// TIA Portal V15 program export: 0 tag tables, 1 data types, 9 data blocks, 101 code blocks (in call order from the OBs), 80 instance data blocks

TYPE "EM_I_OUT_UDT"
// stored: CreationDate 2018-06-03T17:21:19.3788416Z, InterfaceModifiedDate 2018-06-03T17:22:01.3782438Z, IsConsistent true, IsKnowHowProtected false, LibraryConformanceStatus The object is library-conformant., ModifiedDate 2018-06-03T17:22:01.3782438Z
   STRUCT
      Request : Int;
      Command : Int;
      Pressure_SP : REAL;
      placeholder_SP_0 : Byte;   // placeholder
      placeholder_SP_1 : Byte;   // placeholder
      placeholder_SP_2 : Byte;   // placeholder
      placeholder_SP_3 : Byte;   // placeholder
      placeholder_SP_4 : Byte;   // placeholder
      placeholder_SP_5 : Byte;   // placeholder
      placeholder_SP_6 : Byte;   // placeholder
      placeholder_SP_7 : Byte;   // placeholder
      placeholder_SP_8 : Byte;   // placeholder
      placeholder_SP_9 : Byte;   // placeholder
      placeholder_SP_10 : Byte;   // placeholder
      placeholder_SP_11 : Byte;   // placeholder
      placeholder_SP_12 : Byte;   // placeholder
      placeholder_SP_13 : Byte;   // placeholder
      placeholder_SP_14 : Byte;   // placeholder
      placeholder_SP_15 : Byte;   // placeholder
      placeholder_SP_16 : Byte;   // placeholder
      placeholder_SP_17 : Byte;   // placeholder
      placeholder_SP_18 : Byte;   // placeholder
      placeholder_SP_19 : Byte;   // placeholder
      placeholder_SP_20 : Byte;   // placeholder
      placeholder_SP_21 : Byte;   // placeholder
      placeholder_SP_22 : Byte;   // placeholder
      placeholder_SP_23 : Byte;   // placeholder
      placeholder_SP_24 : Byte;   // placeholder
      placeholder_SP_25 : Byte;   // placeholder
      placeholder_SP_26 : Byte;   // placeholder
      placeholder_SP_27 : Byte;   // placeholder
      placeholder_SP_28 : Byte;   // placeholder
      placeholder_SP_29 : Byte;   // placeholder
      placeholder_SP_30 : Byte;   // placeholder
      placeholder_SP_31 : Byte;   // placeholder
      Owner : Int;
      Status : Int;
      CM_error : Bool;
      CM_error_no : DINT;
      q_bACTVIE : Bool;
      Level : REAL;
      Pressure : REAL;
      placeholder_PV_0 : Byte;   // placeholder
      placeholder_PV_1 : Byte;   // placeholder
      placeholder_PV_2 : Byte;   // placeholder
      placeholder_PV_3 : Byte;   // placeholder
      placeholder_PV_4 : Byte;   // placeholder
      placeholder_PV_5 : Byte;   // placeholder
      placeholder_PV_6 : Byte;   // placeholder
      placeholder_PV_7 : Byte;   // placeholder
      placeholder_PV_8 : Byte;   // placeholder
      placeholder_PV_9 : Byte;   // placeholder
      placeholder_PV_10 : Byte;   // placeholder
      placeholder_PV_11 : Byte;   // placeholder
      placeholder_PV_12 : Byte;   // placeholder
      placeholder_PV_13 : Byte;   // placeholder
      placeholder_PV_14 : Byte;   // placeholder
      placeholder_PV_15 : Byte;   // placeholder
      placeholder_PV_16 : Byte;   // placeholder
      placeholder_PV_17 : Byte;   // placeholder
      placeholder_PV_18 : Byte;   // placeholder
      placeholder_PV_19 : Byte;   // placeholder
   END_STRUCT;
END_TYPE

DATA_BLOCK "FIC100_sp"   // DB1
{ S7_Optimized_Access := 'FALSE' }
VERSION : 0.1
// stored: AutoNumber true, CodeModifiedDate 2018-05-31T16:37:51.7325883Z, CompileDate 2018-05-31T16:37:51.7405888Z, CreationDate 2018-05-31T16:36:47.0278874Z, InterfaceModifiedDate 2018-05-31T16:37:42.3500517Z, IsConsistent true, IsKnowHowProtected false, IsOnlyStoredInLoadMemory false, IsPLCDB false, IsWriteProtectedInAS false, ModifiedDate 2018-05-31T16:37:51.7325883Z, ParameterModified 2018-05-31T16:37:42.3500517Z, StructureModified 2018-05-31T16:37:42.3500517Z
   VAR RETAIN
      Operator_Setpoint : Real;
      Set_SP : Bool;
      Output_Value : Real;
      Set_Output : Bool;
   END_VAR
BEGIN
END_DATA_BLOCK

DATA_BLOCK "FIC101_sp"   // DB1
{ S7_Optimized_Access := 'FALSE' }
VERSION : 0.1
// stored: AutoNumber true, CodeModifiedDate 2018-05-31T16:37:51.7325883Z, CompileDate 2018-05-31T16:37:51.7405888Z, CreationDate 2018-05-31T16:36:47.0278874Z, InterfaceModifiedDate 2018-05-31T16:37:42.3500517Z, IsConsistent true, IsKnowHowProtected false, IsOnlyStoredInLoadMemory false, IsPLCDB false, IsWriteProtectedInAS false, ModifiedDate 2018-05-31T16:37:51.7325883Z, ParameterModified 2018-05-31T16:37:42.3500517Z, StructureModified 2018-05-31T16:37:42.3500517Z
   VAR RETAIN
      Operator_Setpoint : Real;
      Set_SP : Bool;
      Output_Value : Real;
      Set_Output : Bool;
   END_VAR
BEGIN
END_DATA_BLOCK

DATA_BLOCK "LIC001_sp"   // DB1
{ S7_Optimized_Access := 'FALSE' }
VERSION : 0.1
// stored: AutoNumber true, CodeModifiedDate 2018-05-31T16:37:51.7325883Z, CompileDate 2018-05-31T16:37:51.7405888Z, CreationDate 2018-05-31T16:36:47.0278874Z, InterfaceModifiedDate 2018-05-31T16:37:42.3500517Z, IsConsistent true, IsKnowHowProtected false, IsOnlyStoredInLoadMemory false, IsPLCDB false, IsWriteProtectedInAS false, ModifiedDate 2018-05-31T16:37:51.7325883Z, ParameterModified 2018-05-31T16:37:42.3500517Z, StructureModified 2018-05-31T16:37:42.3500517Z
   VAR RETAIN
      Operator_Setpoint : Real;
      Set_SP : Bool;
      Output_Value : Real;
      Set_Output : Bool;
   END_VAR
BEGIN
END_DATA_BLOCK

DATA_BLOCK "LIC002_sp"   // DB1
{ S7_Optimized_Access := 'FALSE' }
VERSION : 0.1
// stored: AutoNumber true, CodeModifiedDate 2018-05-31T16:37:51.7325883Z, CompileDate 2018-05-31T16:37:51.7405888Z, CreationDate 2018-05-31T16:36:47.0278874Z, InterfaceModifiedDate 2018-05-31T16:37:42.3500517Z, IsConsistent true, IsKnowHowProtected false, IsOnlyStoredInLoadMemory false, IsPLCDB false, IsWriteProtectedInAS false, ModifiedDate 2018-05-31T16:37:51.7325883Z, ParameterModified 2018-05-31T16:37:42.3500517Z, StructureModified 2018-05-31T16:37:42.3500517Z
   VAR RETAIN
      Operator_Setpoint : Real;
      Set_SP : Bool;
      Output_Value : Real;
      Set_Output : Bool;
   END_VAR
BEGIN
END_DATA_BLOCK

DATA_BLOCK "LIC003_sp"   // DB1
{ S7_Optimized_Access := 'FALSE' }
VERSION : 0.1
// stored: AutoNumber true, CodeModifiedDate 2018-05-31T16:37:51.7325883Z, CompileDate 2018-05-31T16:37:51.7405888Z, CreationDate 2018-05-31T16:36:47.0278874Z, InterfaceModifiedDate 2018-05-31T16:37:42.3500517Z, IsConsistent true, IsKnowHowProtected false, IsOnlyStoredInLoadMemory false, IsPLCDB false, IsWriteProtectedInAS false, ModifiedDate 2018-05-31T16:37:51.7325883Z, ParameterModified 2018-05-31T16:37:42.3500517Z, StructureModified 2018-05-31T16:37:42.3500517Z
   VAR RETAIN
      Operator_Setpoint : Real;
      Set_SP : Bool;
      Output_Value : Real;
      Set_Output : Bool;
   END_VAR
BEGIN
END_DATA_BLOCK

DATA_BLOCK "LIC004_sp"   // DB1
{ S7_Optimized_Access := 'FALSE' }
VERSION : 0.1
// stored: AutoNumber true, CodeModifiedDate 2018-05-31T16:37:51.7325883Z, CompileDate 2018-05-31T16:37:51.7405888Z, CreationDate 2018-05-31T16:36:47.0278874Z, InterfaceModifiedDate 2018-05-31T16:37:42.3500517Z, IsConsistent true, IsKnowHowProtected false, IsOnlyStoredInLoadMemory false, IsPLCDB false, IsWriteProtectedInAS false, ModifiedDate 2018-05-31T16:37:51.7325883Z, ParameterModified 2018-05-31T16:37:42.3500517Z, StructureModified 2018-05-31T16:37:42.3500517Z
   VAR RETAIN
      Operator_Setpoint : Real;
      Set_SP : Bool;
      Output_Value : Real;
      Set_Output : Bool;
   END_VAR
BEGIN
END_DATA_BLOCK

DATA_BLOCK "LIC005_sp"   // DB1
{ S7_Optimized_Access := 'FALSE' }
VERSION : 0.1
// stored: AutoNumber true, CodeModifiedDate 2018-05-31T16:37:51.7325883Z, CompileDate 2018-05-31T16:37:51.7405888Z, CreationDate 2018-05-31T16:36:47.0278874Z, InterfaceModifiedDate 2018-05-31T16:37:42.3500517Z, IsConsistent true, IsKnowHowProtected false, IsOnlyStoredInLoadMemory false, IsPLCDB false, IsWriteProtectedInAS false, ModifiedDate 2018-05-31T16:37:51.7325883Z, ParameterModified 2018-05-31T16:37:42.3500517Z, StructureModified 2018-05-31T16:37:42.3500517Z
   VAR RETAIN
      Operator_Setpoint : Real;
      Set_SP : Bool;
      Output_Value : Real;
      Set_Output : Bool;
   END_VAR
BEGIN
END_DATA_BLOCK

DATA_BLOCK "LIC006_sp"   // DB1
{ S7_Optimized_Access := 'FALSE' }
VERSION : 0.1
// stored: AutoNumber true, CodeModifiedDate 2018-05-31T16:37:51.7325883Z, CompileDate 2018-05-31T16:37:51.7405888Z, CreationDate 2018-05-31T16:36:47.0278874Z, InterfaceModifiedDate 2018-05-31T16:37:42.3500517Z, IsConsistent true, IsKnowHowProtected false, IsOnlyStoredInLoadMemory false, IsPLCDB false, IsWriteProtectedInAS false, ModifiedDate 2018-05-31T16:37:51.7325883Z, ParameterModified 2018-05-31T16:37:42.3500517Z, StructureModified 2018-05-31T16:37:42.3500517Z
   VAR RETAIN
      Operator_Setpoint : Real;
      Set_SP : Bool;
      Output_Value : Real;
      Set_Output : Bool;
   END_VAR
BEGIN
END_DATA_BLOCK

DATA_BLOCK "EM_Index"   // DB2
{ S7_Optimized_Access := 'FALSE' }
VERSION : 0.1
// stored: AutoNumber true, CodeModifiedDate 2018-06-04T11:31:36.2595073Z, CompileDate 2018-06-04T11:31:36.8205394Z, CreationDate 2018-06-04T11:30:27.8755959Z, InterfaceModifiedDate 2018-06-04T11:31:33.0593242Z, IsConsistent true, IsKnowHowProtected false, IsOnlyStoredInLoadMemory false, IsPLCDB false, IsWriteProtectedInAS false, ModifiedDate 2018-06-04T11:31:36.2595073Z, ParameterModified 2018-06-04T11:31:33.0593242Z, StructureModified 2018-06-04T11:31:33.0593242Z
   VAR RETAIN
      DB_Numbers : Array[0..990] of Int;   // DB numbers of the EMs
   END_VAR
BEGIN
END_DATA_BLOCK

ORGANIZATION_BLOCK "Main"   // OB1, STL, ProgramCycle
TITLE = "Main Program Sweep (Cycle)"
{ S7_Optimized_Access := 'FALSE' }
VERSION : 0.1
// stored: AutoNumber false, CodeModifiedDate 2018-06-08T08:01:58.298282Z, CompileDate 2018-06-08T08:01:58.2972819Z, CreationDate 2018-05-29T13:31:39.8908501Z, InterfaceModifiedDate 2007-08-03T16:55:08.419547Z, IsConsistent true, IsKnowHowProtected false, IsWriteProtected false, ModifiedDate 2018-06-08T08:01:58.298282Z, ParameterModified 2007-08-03T16:55:08.419547Z, StructureModified 2007-08-03T16:55:08.419547Z
   VAR_TEMP
      OB1_EV_CLASS : Byte;   // Bits 0-3 = 1 (Coming event), Bits 4-7 = 1 (Event class 1)
      OB1_SCAN_1 : Byte;   // 1 (Cold restart scan 1 of OB 1), 3 (Scan 2-n of OB 1)
      OB1_PRIORITY : Byte;   // Priority of OB Execution
      OB1_OB_NUMBR : Byte;   // 1 (Organization block 1, OB1)
      OB1_RESERVED_1 : Byte;   // Reserved for system
      OB1_RESERVED_2 : Byte;   // Reserved for system
      OB1_PREV_CYCLE : Int;   // Cycle time of previous OB1 scan (milliseconds)
      OB1_MIN_CYCLE : Int;   // Minimum cycle time of OB1 (milliseconds)
      OB1_MAX_CYCLE : Int;   // Maximum cycle time of OB1 (milliseconds)
      OB1_DATE_TIME : Date_And_Time;   // Date and time OB1 started
   END_VAR
BEGIN

NETWORK
TITLE = Main
// comment


      CALL  "Main_Program";


END_ORGANIZATION_BLOCK

FUNCTION "Main_Program" : Void   // FC1, STL
TITLE = Program
{ S7_Optimized_Access := 'TRUE' }
VERSION : 0.1
// Main Program
// stored: AutoNumber true, UDAEnableTagReadback false
BEGIN

NETWORK
TITLE = Main
// comment


      CALL  "Units";

      CALL  "CM_VALVE"
      ( AUT_OP   := ,
        FB_OPEN  := ,
        FB_CLOSE := ,
        QOPEN    := ,
        QCLOSE   := ,
        QMON_ERR := ,
        QCMD_OP  := 
      );



END_FUNCTION

FUNCTION "Units" : Void   // FC1, STL
TITLE = Program
{ S7_Optimized_Access := 'TRUE' }
VERSION : 0.1
// Call all the Units
// stored: AutoNumber true, UDAEnableTagReadback false
BEGIN

NETWORK
TITLE = Main
// comment


// code



END_FUNCTION

FUNCTION_BLOCK "EM_I_OUT"   // FB1, STL
TITLE = EM_I_OUT_fc
{ S7_Optimized_Access := 'TRUE' }
VERSION : 0.1
// EM_I_OUT
// stored: AutoNumber true, UDAEnableTagReadback false
   VAR_INPUT
      sampletime : Real;   // the scantime of this EM/phase, used to increase timers
      em_id : Int;   // undefined - undefined
      Request : Int;   // undefined - undefined
      Command : Int;   // undefined - undefined
      Pressure_SP : REAL;   // undefined - undefined
      Pump_RUN : Bool;   // undefined - undefined
      Pump_QERR : BOOL;   // undefined - General Error
      Pump_EERR : BOOL;   // undefined - External Error
      FS01_PV : Bool;   // Flow Switch - Digital Measurement
      PIC01_PV : REAL;   // Pressure Controller - undefined
      PIC01_ERR : BOOL;   // Pressure Controller - undefined
      LT01_PV : Real;   // Level Transmitter (m) - undefined
      LT01_AHH : Bool;   // Level Transmitter (m) - undefined
      LT01_AH : Bool;   // Level Transmitter (m) - undefined
      LT01_AL : Bool;   // Level Transmitter (m) - undefined
      LT01_ALL : Bool;   // Level Transmitter (m) - undefined
      LT01_ERR : BOOL;   // Level Transmitter (m) - undefined
      XV_Bottom_OPN : BOOL;   // Automatic Bottom Valve - undefined
      XV_Bottom_CLS : BOOL;   // Automatic Bottom Valve - undefined
      XV_Bottom_MERR : BOOL;   // Automatic Bottom Valve - undefined
      BV_Bottom_OPN : BOOL;   // Manual Bottom Valve - undefined
      BV_Bottom_CLS : BOOL;   // Manual Bottom Valve - undefined
      BV_Bottom_MERR : BOOL;   // Manual Bottom Valve - undefined
      BV_Tran_M04_OPN : BOOL;   // Trnasfer Valve to M04 - undefined
      BV_Tran_M04_CLS : BOOL;   // Trnasfer Valve to M04 - undefined
      BV_Tran_M04_MERR : BOOL;   // Trnasfer Valve to M04 - undefined
   END_VAR
   VAR_OUTPUT
      steptime_s : Real;   // complete steptime in seconds. same value as the other steptimes
      steptime_m : Real;   // complete steptime in minutes. same value as the other steptimes
      steptime_h : Real;   // complete steptime in hours. same value as the other steptimes
      first_scan : Bool;   // first scan of the step active
      last_scan : Bool;   // last scan of the step active
      error_index_db : Bool;   // em_id doesn't fit in the index db
      Owner : Int;   // undefined - undefined
      Status : Int;   // undefined - undefined
      CM_error : Bool;   // undefined - undefined
      CM_error_no : DINT;   // undefined - undefined
      q_bACTVIE : Bool;   // undefined - undefined
      Level : REAL;   // undefined - undefined
      Pressure : REAL;   // undefined - undefined
      Pump_ON : Bool;   // undefined - Switch Motor ON
      Pump_AUT : Bool;   // undefined - Swtich Motor to AUTO
      PIC01_EXT : Bool;   // Pressure Controller - Switch to External Mode
      PIC01_SP : Real;   // Pressure Controller - Operator Setpoint in Internal Mode
      PIC01_AUT : Bool;   // Pressure Controller - Switch to Auto Mode
      PIC01_VAL_OUT : Real;   // Pressure Controller - Operator Output Value
      PIC01_SET_SP : Bool;   // Pressure Controller - undefined
      PIC01_SET_OUT : Bool;   // Pressure Controller - undefined
      XV_Bottom_CMD : BOOL;   // Automatic Bottom Valve - Auto command from program
      BV_Bottom_CMD : BOOL;   // Manual Bottom Valve - Auto command from program
      BV_Tran_M04_CMD : BOOL;   // Trnasfer Valve to M04 - Auto command from program
   END_VAR
   VAR DB_SPECIFIC
      previous_Command : Int;   // previous Command
      SP_PV : "EM_I_OUT_UDT";   // UDT for receiving Setpoints and sending Process Values
   END_VAR
   VAR_TEMP
      initial_scan : Bool;   // pulse active on the first cycle of a new scan
      T_dbnum : Int;   // DB number of this block
      T_address : Int;   // address in the Index Table DB
      T_length : Int;   // length of the Index Table DB
   END_VAR
BEGIN

NETWORK
TITLE = Publish DB number to EM Index
// The EM will publish its DB number to the EM Index table


//### 0] init
      CLR;
      =     #error_index_db;


//### 1] Check if the ID of this EM fits inside the EM Index table

      OPN   "EM_Index";  //Open data block as shared data block
      L     DBLG;  //Load length of shared data block (length of DB)
      T     #T_length;  //transfer length to length

      L     #T_length;  //length=length/2
      L     2;
      /I;
      T     #T_length;

// Error and end the block if id bigger than length of the DB
      L     #T_length;
      L     #em_id;
      <=D;
      =     #error_index_db;
      BEC;  //if id is bigger than length end the block

//### 2] Write this DB number to the EM Index table

// find the number of the current fb
      L     DINO;
      T     #T_dbnum;  //find the db number of current fb

// calculate the real address
      L     #em_id;
      L     2;
      *I;
      T     #T_address;

// prepare the pointer for the location in the EM Index DB
// todo: can this code not simpeler? Probably no need to add with the zero-pointer
      OPN   "EM_Index";
      L     P#DBX0.0;
      L     #T_address;
      SLD   3;
      +D;
      LAR1;

//write the DB number to the real address
      L     #T_dbnum;
      T     DBW [AR1, P#0.0];





NETWORK
TITLE = Copy all Setpoints from the UDT
// network comment





      L     #SP_PV.Request;
      T     #Request;



      L     #SP_PV.Command;
      T     #Command;



      L     #SP_PV.Pressure_SP;
      T     #Pressure_SP;




NETWORK
TITLE = Acquiring logic
// network comment


      L     #Request;
      T     #Owner;



NETWORK
TITLE = Steptimers
// If the previous Command is not the same as the current one
// then reset the timers, else increase them
// This is at the start of the FB because normal commandchanges will take
// till the next cycle to become active


// check if Command == previous_Command
      L     #Command;
      L     #previous_Command;
      ==I;  //if condition true then {
      JCN   TIM1;

// increase timer
      L     #sampletime;
      L     #steptime_s;
      +R;
      T     #steptime_s;

      JU    TIM2;
TIM1: NOP   0;

// reset timer
      L     0.0;
      T     #steptime_s;

TIM2: NOP   0;  //end if

// calculate the other two timers
      L     #steptime_s;
      L     60.0;
      /R;
      T     #steptime_m;

      L     60.0;
      /R;
      T     #steptime_h;



NETWORK
TITLE = detect initial scan
// create a pulse active on the first cycle of a new scan
// this signal can be used in the state to execute some actions in the first cycle of the state


      L     #Command;
      L     #previous_Command;
      <>I;
      =     #initial_scan;



NETWORK
TITLE = Save old step
// network comment


      L     #Command;
      T     #previous_Command;



NETWORK
TITLE = Collect the errors from the CMs
// network comment


      CLR;
      O     #Pump_QERR;
      O     #Pump_EERR;
      O     #PIC01_ERR;
      O     #LT01_ERR;
      O     #XV_Bottom_MERR;
      O     #BV_Bottom_MERR;
      O     #BV_Tran_M04_MERR;
      =     #CM_error;



NETWORK
TITLE = Assign a message number to each error
// This code tries to assign an error message to each CM error
// If multiple CMs have an error then it only stores one
// This is the EM type so we don't know which CM instance is connected
// So the error only contains the general name of the CM instance
// If the actual name needs to be shown then it could be deducted
// at a higher level using the CM name and EM instance 
// network_end.render(lib, "ssign a message number to each error") }}


      CLR;

// clear the error no
      L     0;
      T     #CM_error_no;



      A     #Pump_QERR;
      JCN   E1;

      L     50;  //'CM error: Pump_QERR'
      T     #CM_error_no;

E1:   NOP   0;

      A     #Pump_EERR;
      JCN   E2;

      L     51;  //'CM error: Pump_EERR'
      T     #CM_error_no;

E2:   NOP   0;

      A     #PIC01_ERR;
      JCN   E3;

      L     52;  //'CM error: PIC01_ERR'
      T     #CM_error_no;

E3:   NOP   0;

      A     #LT01_ERR;
      JCN   E4;

      L     53;  //'CM error: LT01_ERR'
      T     #CM_error_no;

E4:   NOP   0;

      A     #XV_Bottom_MERR;
      JCN   E5;

      L     54;  //'CM error: XV_Bottom_MERR'
      T     #CM_error_no;

E5:   NOP   0;

      A     #BV_Bottom_MERR;
      JCN   E6;

      L     55;  //'CM error: BV_Bottom_MERR'
      T     #CM_error_no;

E6:   NOP   0;

      A     #BV_Tran_M04_MERR;
      JCN   E7;

      L     56;  //'CM error: BV_Tran_M04_MERR'
      T     #CM_error_no;

E7:   NOP   0;



NETWORK
TITLE = START OF THE STATES
// ################################
// ################################
// 	Placeholder network to indicate the start of the actual sequence
// ################################	  
// ################################


// empty placeholder network



NETWORK
TITLE = State 0: undefined


// skip this network if stepnumber not equal to 0
      L     #Command;
      L     0;
      ==I;
      JCN   J1;

//---------------------------------
// Actions (continuous)
//---------------------------------

// Action: stop Pump
      CLR;
      =     #Pump_ON;

// Action: close XV_Bottom
      CLR;
      =     #XV_Bottom_CMD;

// Action: close BV_Bottom
      CLR;
      =     #BV_Bottom_CMD;

// Action: close BV_Tran_M04
      CLR;
      =     #BV_Tran_M04_CMD;
//---------------------------------
// --- CONDITIONS ---
//---------------------------------

// Condition Logic
      SET;  //make sure RLO is high so the state can happen when no conditions present

      A     #XV_Bottom_CLS;  //XV_Bottom close
      A     #BV_Bottom_CLS;  //BV_Bottom close
      A     #BV_Tran_M04_CLS;  //BV_Tran_M04 close
      JCN   L1;

      L     #Command;
      T     #Status;

L1:   NOP   0;

D1:   NOP   0;

//---------------------------------
// End of network: jump here if step not active
// Jump to end of this FB if the step has been active to avoid
// execution of another step in the same scan
//---------------------------------
      JU    ENDS;
J1:   NOP   0;




NETWORK
TITLE = State 1: undefined


// skip this network if stepnumber not equal to 1
      L     #Command;
      L     1;
      ==I;
      JCN   J2;

//---------------------------------
// Actions (continuous)
//---------------------------------

// Action: stop Pump
      CLR;
      =     #Pump_ON;

// Action: open XV_Bottom
      SET;
      =     #XV_Bottom_CMD;
//---------------------------------
// --- CONDITIONS ---
//---------------------------------

// Condition Logic
      SET;  //make sure RLO is high so the state can happen when no conditions present

      A     #XV_Bottom_OPN;  //XV_Bottom open
      JCN   L2;

      L     #Command;
      T     #Status;

L2:   NOP   0;

D2:   NOP   0;

//---------------------------------
// End of network: jump here if step not active
// Jump to end of this FB if the step has been active to avoid
// execution of another step in the same scan
//---------------------------------
      JU    ENDS;
J2:   NOP   0;




NETWORK
TITLE = State 2: undefined


// skip this network if stepnumber not equal to 2
      L     #Command;
      L     2;
      ==I;
      JCN   J3;

//---------------------------------
// Actions (first scan)
//---------------------------------
      A     #initial_scan;
      JCN   C3;
      L     -1.0;  //value to show that the EM is in a state transition
      T     #Status;

// Action: PIC01_SP = 10.0
      L     10.0;
      T     #PIC01_SP;

// Action: PIC01_SET_SP = true
      SET;
      =     #PIC01_SET_SP;

      JU    D3;
C3:   NOP   0;


//---------------------------------
// Actions (continuous)
//---------------------------------

// Action: start Pump
      SET;
      =     #Pump_ON;

// Action: auto 10.0 bar PIC01
      SET;
      =     #PIC01_AUT;

// Action: open XV_Bottom
      SET;
      =     #XV_Bottom_CMD;

// Action: PIC01_SET_SP = false
      CLR;
      =     #PIC01_SET_SP;
//---------------------------------
// --- CONDITIONS ---
//---------------------------------

// Condition Logic
      SET;  //make sure RLO is high so the state can happen when no conditions present

      A     #Pump_RUN;  //Pump start
      A     #XV_Bottom_OPN;  //XV_Bottom open
      JCN   L3;

      L     #Command;
      T     #Status;

L3:   NOP   0;

D3:   NOP   0;

//---------------------------------
// End of network: jump here if step not active
// Jump to end of this FB if the step has been active to avoid
// execution of another step in the same scan
//---------------------------------
      JU    ENDS;
J3:   NOP   0;




NETWORK
TITLE = State 3: undefined


// skip this network if stepnumber not equal to 3
      L     #Command;
      L     3;
      ==I;
      JCN   J4;

//---------------------------------
// Actions (continuous)
//---------------------------------

// Action: stop Pump
      CLR;
      =     #Pump_ON;

// Action: open BV_Bottom
      SET;
      =     #BV_Bottom_CMD;

// Action: open BV_Tran_M04
      SET;
      =     #BV_Tran_M04_CMD;
//---------------------------------
// --- CONDITIONS ---
//---------------------------------

// Condition Logic
      SET;  //make sure RLO is high so the state can happen when no conditions present

      A     #BV_Bottom_OPN;  //BV_Bottom open
      A     #BV_Tran_M04_OPN;  //BV_Tran_M04 open
      JCN   L4;

      L     #Command;
      T     #Status;

L4:   NOP   0;

D4:   NOP   0;

//---------------------------------
// End of network: jump here if step not active
// Jump to end of this FB if the step has been active to avoid
// execution of another step in the same scan
//---------------------------------
      JU    ENDS;
J4:   NOP   0;




NETWORK
TITLE = State 4: undefined


// skip this network if stepnumber not equal to 4
      L     #Command;
      L     4;
      ==I;
      JCN   J5;

//---------------------------------
// Actions (first scan)
//---------------------------------
      A     #initial_scan;
      JCN   C5;
      L     -1.0;  //value to show that the EM is in a state transition
      T     #Status;

// Action: PIC01_SP = Pressure_SP
      L     #Pressure_SP;
      T     #PIC01_SP;

// Action: PIC01_SET_SP = true
      SET;
      =     #PIC01_SET_SP;

      JU    D5;
C5:   NOP   0;


//---------------------------------
// Actions (continuous)
//---------------------------------

// Action: start Pump
      SET;
      =     #Pump_ON;

// Action: auto Pressure_SP PIC01
      SET;
      =     #PIC01_AUT;

// Action: open BV_Bottom
      SET;
      =     #BV_Bottom_CMD;

// Action: open BV_Tran_M04
      SET;
      =     #BV_Tran_M04_CMD;

// Action: PIC01_SET_SP = false
      CLR;
      =     #PIC01_SET_SP;
//---------------------------------
// --- CONDITIONS ---
//---------------------------------

// Condition Logic
      SET;  //make sure RLO is high so the state can happen when no conditions present

      A     #Pump_RUN;  //Pump start
      A     #BV_Bottom_OPN;  //BV_Bottom open
      A     #BV_Tran_M04_OPN;  //BV_Tran_M04 open
      JCN   L5;

      L     #Command;
      T     #Status;

L5:   NOP   0;

D5:   NOP   0;

//---------------------------------
// End of network: jump here if step not active
// Jump to end of this FB if the step has been active to avoid
// execution of another step in the same scan
//---------------------------------
      JU    ENDS;
J5:   NOP   0;




NETWORK
TITLE = State 5: undefined


// skip this network if stepnumber not equal to 5
      L     #Command;
      L     5;
      ==I;
      JCN   J6;

//---------------------------------
// Actions (first scan)
//---------------------------------
      A     #initial_scan;
      JCN   C6;
      L     -1.0;  //value to show that the EM is in a state transition
      T     #Status;

// Action: PIC01_VAL_OUT = 20.0
      L     20.0;
      T     #PIC01_VAL_OUT;

// Action: PIC01_SET_OUT = true
      SET;
      =     #PIC01_SET_OUT;

      JU    D6;
C6:   NOP   0;


//---------------------------------
// Actions (continuous)
//---------------------------------

// Action: start Pump
      SET;
      =     #Pump_ON;

// Action: manual 20.0 Hz PIC01
      CLR;
      =     #PIC01_AUT;

// Action: open XV_Bottom
      SET;
      =     #XV_Bottom_CMD;

// Action: PIC01_SET_OUT = false
      CLR;
      =     #PIC01_SET_OUT;
//---------------------------------
// --- CONDITIONS ---
//---------------------------------

// Condition Logic
      SET;  //make sure RLO is high so the state can happen when no conditions present

      A     #Pump_RUN;  //Pump start
      A     #XV_Bottom_OPN;  //XV_Bottom open
      JCN   L6;

      L     #Command;
      T     #Status;

L6:   NOP   0;

D6:   NOP   0;

//---------------------------------
// End of network: jump here if step not active
// Jump to end of this FB if the step has been active to avoid
// execution of another step in the same scan
//---------------------------------
      JU    ENDS;
J6:   NOP   0;




NETWORK
TITLE = END OF THE STATES
// ################################
// ################################
// 	Placeholder network to indicate the end of the actual sequence
// ################################	  
// ################################


// jump location for the state that is currently active
ENDS: NOP   0;



NETWORK
TITLE = eneral Actions - After
// General Actions - After


// Action: Level = LT01
      L     #LT01_PV;
      T     #Level;

// Action: Pressure = PIC01
      L     #PIC01_PV;
      T     #Pressure;


NETWORK
TITLE = Copy all Process Values to the UDT
// network comment





      L     #Owner;
      T     #SP_PV.Owner;



      L     #Status;
      T     #SP_PV.Status;



      A     #CM_error;
      =     #SP_PV.CM_error;



      L     #CM_error_no;
      T     #SP_PV.CM_error_no;



      A     #q_bACTVIE;
      =     #SP_PV.q_bACTVIE;



      L     #Level;
      T     #SP_PV.Level;



      L     #Pressure;
      T     #SP_PV.Pressure;




NETWORK
TITLE = Clean up request
// Phases don't clean up their requests on the EM side
// So at the end of the EM reset the request
// If the phase is still there then it will write the request again by the next scan


      L     0;
      T     "request";



NETWORK
TITLE = network title
// network comment


// empty placeholder network


END_FUNCTION_BLOCK

FUNCTION "EM_Instance_10_fc" : Void   // FC1, STL
TITLE = _fc
{ S7_Optimized_Access := 'TRUE' }
VERSION : 0.1
// test
// stored: AutoNumber true, UDAEnableTagReadback false
BEGIN

NETWORK
TITLE = Main
// comment:


// Call the EM FB with the corresponding DB instance
      CALL  "EM_I_OUT", "EM_Instance_10"
      ( sampletime       := ,
        em_id            := 35,
        Request          := ,
        Command          := ,
        Pressure_SP      := ,
        Pump_RUN         := "M106".QNOFF2,
        Pump_QERR        := "M106".QERR,
        Pump_EERR        := "M106".QERR_EXT,
        FS01_PV          := "LS002".QON,
        PIC01_PV         := "FIC101".PV,
        PIC01_ERR        := "FIC101".QERR,
        LT01_PV          := "LT101".QfVal,
        LT01_AHH         := "LT101".LIM_Qb01,
        LT01_AH          := "LT101".LIM_Qb02,
        LT01_AL          := "LT101".LIM_Qb03,
        LT01_ALL         := "LT101".LIM_Qb04,
        LT01_ERR         := "LT101".QERR,
        XV_Bottom_OPN    := ,
        XV_Bottom_CLS    := ,
        XV_Bottom_MERR   := ,
        BV_Bottom_OPN    := "MV007".QOPEN,
        BV_Bottom_CLS    := "MV007".QCLOSE,
        BV_Bottom_MERR   := "MV007".QMON_ERR,
        BV_Tran_M04_OPN  := ,
        BV_Tran_M04_CLS  := ,
        BV_Tran_M04_MERR := ,
        steptime_s       := ,
        steptime_m       := ,
        steptime_h       := ,
        first_scan       := ,
        last_scan        := ,
        error_index_db   := ,
        Owner            := ,
        Status           := ,
        CM_error         := ,
        CM_error_no      := ,
        q_bACTVIE        := ,
        Level            := ,
        Pressure         := ,
        Pump_ON          := "M106".L_ON,
        Pump_AUT         := "M106".L_AUT,
        PIC01_EXT        := "FIC101".L_REMOTE,
        PIC01_SP         := "FIC101".HMI_SP_INT,
        PIC01_AUT        := "FIC101".L_AUT,
        PIC01_VAL_OUT    := "FIC101".HMI_MAN,
        PIC01_SET_SP     := "FIC101".Set_SP,
        PIC01_SET_OUT    := "FIC101".Set_Output,
        XV_Bottom_CMD    := ,
        BV_Bottom_CMD    := "MV007".AUT_OP,
        BV_Tran_M04_CMD  := 
      );
END_FUNCTION

FUNCTION "EM_Instance_11_fc" : Void   // FC1, STL
TITLE = _fc
{ S7_Optimized_Access := 'TRUE' }
VERSION : 0.1
// test
// stored: AutoNumber true, UDAEnableTagReadback false
BEGIN

NETWORK
TITLE = Main
// comment:


// Call the EM FB with the corresponding DB instance
      CALL  "EM_I_OUT", "EM_Instance_11"
      ( sampletime       := ,
        em_id            := 36,
        Request          := ,
        Command          := ,
        Pressure_SP      := ,
        Pump_RUN         := "M106".QNOFF2,
        Pump_QERR        := "M106".QERR,
        Pump_EERR        := "M106".QERR_EXT,
        FS01_PV          := "LS002".QON,
        PIC01_PV         := "FIC101".PV,
        PIC01_ERR        := "FIC101".QERR,
        LT01_PV          := "LT201".QfVal,
        LT01_AHH         := "LT201".LIM_Qb01,
        LT01_AH          := "LT201".LIM_Qb02,
        LT01_AL          := "LT201".LIM_Qb03,
        LT01_ALL         := "LT201".LIM_Qb04,
        LT01_ERR         := "LT201".QERR,
        XV_Bottom_OPN    := "XV001".QOPEN,
        XV_Bottom_CLS    := "XV001".QCLOSE,
        XV_Bottom_MERR   := "XV001".QMON_ERR,
        BV_Bottom_OPN    := ,
        BV_Bottom_CLS    := ,
        BV_Bottom_MERR   := ,
        BV_Tran_M04_OPN  := ,
        BV_Tran_M04_CLS  := ,
        BV_Tran_M04_MERR := ,
        steptime_s       := ,
        steptime_m       := ,
        steptime_h       := ,
        first_scan       := ,
        last_scan        := ,
        error_index_db   := ,
        Owner            := ,
        Status           := ,
        CM_error         := ,
        CM_error_no      := ,
        q_bACTVIE        := ,
        Level            := ,
        Pressure         := ,
        Pump_ON          := "M106".L_ON,
        Pump_AUT         := "M106".L_AUT,
        PIC01_EXT        := "FIC101".L_REMOTE,
        PIC01_SP         := "FIC101".HMI_SP_INT,
        PIC01_AUT        := "FIC101".L_AUT,
        PIC01_VAL_OUT    := "FIC101".HMI_MAN,
        PIC01_SET_SP     := "FIC101".Set_SP,
        PIC01_SET_OUT    := "FIC101".Set_Output,
        XV_Bottom_CMD    := "XV001".AUT_OP,
        BV_Bottom_CMD    := ,
        BV_Tran_M04_CMD  := 
      );
END_FUNCTION

FUNCTION "EM_Instance_12_fc" : Void   // FC1, STL
TITLE = _fc
{ S7_Optimized_Access := 'TRUE' }
VERSION : 0.1
// test
// stored: AutoNumber true, UDAEnableTagReadback false
BEGIN

NETWORK
TITLE = Main
// comment:


// Call the EM FB with the corresponding DB instance
      CALL  "EM_I_OUT", "EM_Instance_12"
      ( sampletime       := ,
        em_id            := 37,
        Request          := ,
        Command          := ,
        Pressure_SP      := ,
        Pump_RUN         := "M106".QNOFF2,
        Pump_QERR        := "M106".QERR,
        Pump_EERR        := "M106".QERR_EXT,
        FS01_PV          := "LS002".QON,
        PIC01_PV         := "FIC101".PV,
        PIC01_ERR        := "FIC101".QERR,
        LT01_PV          := "LT201".QfVal,
        LT01_AHH         := "LT201".LIM_Qb01,
        LT01_AH          := "LT201".LIM_Qb02,
        LT01_AL          := "LT201".LIM_Qb03,
        LT01_ALL         := "LT201".LIM_Qb04,
        LT01_ERR         := "LT201".QERR,
        XV_Bottom_OPN    := "XV002".QOPEN,
        XV_Bottom_CLS    := "XV002".QCLOSE,
        XV_Bottom_MERR   := "XV002".QMON_ERR,
        BV_Bottom_OPN    := ,
        BV_Bottom_CLS    := ,
        BV_Bottom_MERR   := ,
        BV_Tran_M04_OPN  := ,
        BV_Tran_M04_CLS  := ,
        BV_Tran_M04_MERR := ,
        steptime_s       := ,
        steptime_m       := ,
        steptime_h       := ,
        first_scan       := ,
        last_scan        := ,
        error_index_db   := ,
        Owner            := ,
        Status           := ,
        CM_error         := ,
        CM_error_no      := ,
        q_bACTVIE        := ,
        Level            := ,
        Pressure         := ,
        Pump_ON          := "M106".L_ON,
        Pump_AUT         := "M106".L_AUT,
        PIC01_EXT        := "FIC101".L_REMOTE,
        PIC01_SP         := "FIC101".HMI_SP_INT,
        PIC01_AUT        := "FIC101".L_AUT,
        PIC01_VAL_OUT    := "FIC101".HMI_MAN,
        PIC01_SET_SP     := "FIC101".Set_SP,
        PIC01_SET_OUT    := "FIC101".Set_Output,
        XV_Bottom_CMD    := "XV002".AUT_OP,
        BV_Bottom_CMD    := ,
        BV_Tran_M04_CMD  := 
      );
END_FUNCTION

FUNCTION "EM_Instance_13_fc" : Void   // FC1, STL
TITLE = _fc
{ S7_Optimized_Access := 'TRUE' }
VERSION : 0.1
// test
// stored: AutoNumber true, UDAEnableTagReadback false
BEGIN

NETWORK
TITLE = Main
// comment:


// Call the EM FB with the corresponding DB instance
      CALL  "EM_I_OUT", "EM_Instance_13"
      ( sampletime       := ,
        em_id            := 38,
        Request          := ,
        Command          := ,
        Pressure_SP      := ,
        Pump_RUN         := "M106".QNOFF2,
        Pump_QERR        := "M106".QERR,
        Pump_EERR        := "M106".QERR_EXT,
        FS01_PV          := "LS002".QON,
        PIC01_PV         := "FIC101".PV,
        PIC01_ERR        := "FIC101".QERR,
        LT01_PV          := "LT201".QfVal,
        LT01_AHH         := "LT201".LIM_Qb01,
        LT01_AH          := "LT201".LIM_Qb02,
        LT01_AL          := "LT201".LIM_Qb03,
        LT01_ALL         := "LT201".LIM_Qb04,
        LT01_ERR         := "LT201".QERR,
        XV_Bottom_OPN    := "XV003".QOPEN,
        XV_Bottom_CLS    := "XV003".QCLOSE,
        XV_Bottom_MERR   := "XV003".QMON_ERR,
        BV_Bottom_OPN    := ,
        BV_Bottom_CLS    := ,
        BV_Bottom_MERR   := ,
        BV_Tran_M04_OPN  := ,
        BV_Tran_M04_CLS  := ,
        BV_Tran_M04_MERR := ,
        steptime_s       := ,
        steptime_m       := ,
        steptime_h       := ,
        first_scan       := ,
        last_scan        := ,
        error_index_db   := ,
        Owner            := ,
        Status           := ,
        CM_error         := ,
        CM_error_no      := ,
        q_bACTVIE        := ,
        Level            := ,
        Pressure         := ,
        Pump_ON          := "M106".L_ON,
        Pump_AUT         := "M106".L_AUT,
        PIC01_EXT        := "FIC101".L_REMOTE,
        PIC01_SP         := "FIC101".HMI_SP_INT,
        PIC01_AUT        := "FIC101".L_AUT,
        PIC01_VAL_OUT    := "FIC101".HMI_MAN,
        PIC01_SET_SP     := "FIC101".Set_SP,
        PIC01_SET_OUT    := "FIC101".Set_Output,
        XV_Bottom_CMD    := "XV003".AUT_OP,
        BV_Bottom_CMD    := ,
        BV_Tran_M04_CMD  := 
      );
END_FUNCTION

FUNCTION "EM_Instance_14_fc" : Void   // FC1, STL
TITLE = _fc
{ S7_Optimized_Access := 'TRUE' }
VERSION : 0.1
// test
// stored: AutoNumber true, UDAEnableTagReadback false
BEGIN

NETWORK
TITLE = Main
// comment:


// Call the EM FB with the corresponding DB instance
      CALL  "EM_I_OUT", "EM_Instance_14"
      ( sampletime       := ,
        em_id            := 39,
        Request          := ,
        Command          := ,
        Pressure_SP      := ,
        Pump_RUN         := "M106".QNOFF2,
        Pump_QERR        := "M106".QERR,
        Pump_EERR        := "M106".QERR_EXT,
        FS01_PV          := "LS002".QON,
        PIC01_PV         := "FIC101".PV,
        PIC01_ERR        := "FIC101".QERR,
        LT01_PV          := "LT201".QfVal,
        LT01_AHH         := "LT201".LIM_Qb01,
        LT01_AH          := "LT201".LIM_Qb02,
        LT01_AL          := "LT201".LIM_Qb03,
        LT01_ALL         := "LT201".LIM_Qb04,
        LT01_ERR         := "LT201".QERR,
        XV_Bottom_OPN    := "XV004".QOPEN,
        XV_Bottom_CLS    := "XV004".QCLOSE,
        XV_Bottom_MERR   := "XV004".QMON_ERR,
        BV_Bottom_OPN    := ,
        BV_Bottom_CLS    := ,
        BV_Bottom_MERR   := ,
        BV_Tran_M04_OPN  := ,
        BV_Tran_M04_CLS  := ,
        BV_Tran_M04_MERR := ,
        steptime_s       := ,
        steptime_m       := ,
        steptime_h       := ,
        first_scan       := ,
        last_scan        := ,
        error_index_db   := ,
        Owner            := ,
        Status           := ,
        CM_error         := ,
        CM_error_no      := ,
        q_bACTVIE        := ,
        Level            := ,
        Pressure         := ,
        Pump_ON          := "M106".L_ON,
        Pump_AUT         := "M106".L_AUT,
        PIC01_EXT        := "FIC101".L_REMOTE,
        PIC01_SP         := "FIC101".HMI_SP_INT,
        PIC01_AUT        := "FIC101".L_AUT,
        PIC01_VAL_OUT    := "FIC101".HMI_MAN,
        PIC01_SET_SP     := "FIC101".Set_SP,
        PIC01_SET_OUT    := "FIC101".Set_Output,
        XV_Bottom_CMD    := "XV004".AUT_OP,
        BV_Bottom_CMD    := ,
        BV_Tran_M04_CMD  := 
      );
END_FUNCTION

FUNCTION "EM_Instance_1_fc" : Void   // FC1, STL
TITLE = _fc
{ S7_Optimized_Access := 'TRUE' }
VERSION : 0.1
// test
// stored: AutoNumber true, UDAEnableTagReadback false
BEGIN

NETWORK
TITLE = Main
// comment:


// Call the EM FB with the corresponding DB instance
      CALL  "EM_I_OUT", "EM_Instance_1"
      ( sampletime       := ,
        em_id            := 26,
        Request          := ,
        Command          := ,
        Pressure_SP      := ,
        Pump_RUN         := "M100".QNOFF2,
        Pump_QERR        := "M100".QERR,
        Pump_EERR        := "M100".QERR_EXT,
        FS01_PV          := "LS001".QON,
        PIC01_PV         := "LIC001".PV,
        PIC01_ERR        := "LIC001".QERR,
        LT01_PV          := "LT001".QfVal,
        LT01_AHH         := "LT001".LIM_Qb01,
        LT01_AH          := "LT001".LIM_Qb02,
        LT01_AL          := "LT001".LIM_Qb03,
        LT01_ALL         := "LT001".LIM_Qb04,
        LT01_ERR         := "LT001".QERR,
        XV_Bottom_OPN    := ,
        XV_Bottom_CLS    := ,
        XV_Bottom_MERR   := ,
        BV_Bottom_OPN    := "MV001".QOPEN,
        BV_Bottom_CLS    := "MV001".QCLOSE,
        BV_Bottom_MERR   := "MV001".QMON_ERR,
        BV_Tran_M04_OPN  := "MV003".QOPEN,
        BV_Tran_M04_CLS  := "MV003".QCLOSE,
        BV_Tran_M04_MERR := "MV003".QMON_ERR,
        steptime_s       := ,
        steptime_m       := ,
        steptime_h       := ,
        first_scan       := ,
        last_scan        := ,
        error_index_db   := ,
        Owner            := ,
        Status           := ,
        CM_error         := ,
        CM_error_no      := ,
        q_bACTVIE        := ,
        Level            := ,
        Pressure         := ,
        Pump_ON          := "M100".L_ON,
        Pump_AUT         := "M100".L_AUT,
        PIC01_EXT        := "LIC001".L_REMOTE,
        PIC01_SP         := "LIC001".HMI_SP_INT,
        PIC01_AUT        := "LIC001".L_AUT,
        PIC01_VAL_OUT    := "LIC001".HMI_MAN,
        PIC01_SET_SP     := "LIC001".Set_SP,
        PIC01_SET_OUT    := "LIC001".Set_Output,
        XV_Bottom_CMD    := ,
        BV_Bottom_CMD    := "MV001".AUT_OP,
        BV_Tran_M04_CMD  := "MV003".AUT_OP
      );
END_FUNCTION

FUNCTION "EM_Instance_2_fc" : Void   // FC1, STL
TITLE = _fc
{ S7_Optimized_Access := 'TRUE' }
VERSION : 0.1
// test
// stored: AutoNumber true, UDAEnableTagReadback false
BEGIN

NETWORK
TITLE = Main
// comment:


// Call the EM FB with the corresponding DB instance
      CALL  "EM_I_OUT", "EM_Instance_2"
      ( sampletime       := ,
        em_id            := 27,
        Request          := ,
        Command          := ,
        Pressure_SP      := ,
        Pump_RUN         := "M101".QNOFF2,
        Pump_QERR        := "M101".QERR,
        Pump_EERR        := "M101".QERR_EXT,
        FS01_PV          := "LS002".QON,
        PIC01_PV         := "LIC002".PV,
        PIC01_ERR        := "LIC002".QERR,
        LT01_PV          := "LT002".QfVal,
        LT01_AHH         := "LT002".LIM_Qb01,
        LT01_AH          := "LT002".LIM_Qb02,
        LT01_AL          := "LT002".LIM_Qb03,
        LT01_ALL         := "LT002".LIM_Qb04,
        LT01_ERR         := "LT002".QERR,
        XV_Bottom_OPN    := ,
        XV_Bottom_CLS    := ,
        XV_Bottom_MERR   := ,
        BV_Bottom_OPN    := "MV002".QOPEN,
        BV_Bottom_CLS    := "MV002".QCLOSE,
        BV_Bottom_MERR   := "MV002".QMON_ERR,
        BV_Tran_M04_OPN  := "MV003".QOPEN,
        BV_Tran_M04_CLS  := "MV003".QCLOSE,
        BV_Tran_M04_MERR := "MV003".QMON_ERR,
        steptime_s       := ,
        steptime_m       := ,
        steptime_h       := ,
        first_scan       := ,
        last_scan        := ,
        error_index_db   := ,
        Owner            := ,
        Status           := ,
        CM_error         := ,
        CM_error_no      := ,
        q_bACTVIE        := ,
        Level            := ,
        Pressure         := ,
        Pump_ON          := "M101".L_ON,
        Pump_AUT         := "M101".L_AUT,
        PIC01_EXT        := "LIC002".L_REMOTE,
        PIC01_SP         := "LIC002".HMI_SP_INT,
        PIC01_AUT        := "LIC002".L_AUT,
        PIC01_VAL_OUT    := "LIC002".HMI_MAN,
        PIC01_SET_SP     := "LIC002".Set_SP,
        PIC01_SET_OUT    := "LIC002".Set_Output,
        XV_Bottom_CMD    := ,
        BV_Bottom_CMD    := "MV002".AUT_OP,
        BV_Tran_M04_CMD  := "MV003".AUT_OP
      );
END_FUNCTION

FUNCTION "EM_Instance_3_fc" : Void   // FC1, STL
TITLE = _fc
{ S7_Optimized_Access := 'TRUE' }
VERSION : 0.1
// test
// stored: AutoNumber true, UDAEnableTagReadback false
BEGIN

NETWORK
TITLE = Main
// comment:


// Call the EM FB with the corresponding DB instance
      CALL  "EM_I_OUT", "EM_Instance_3"
      ( sampletime       := ,
        em_id            := 28,
        Request          := ,
        Command          := ,
        Pressure_SP      := ,
        Pump_RUN         := "M102".QNOFF2,
        Pump_QERR        := "M102".QERR,
        Pump_EERR        := "M102".QERR_EXT,
        FS01_PV          := "LS002".QON,
        PIC01_PV         := "LIC003".PV,
        PIC01_ERR        := "LIC003".QERR,
        LT01_PV          := "LT003".QfVal,
        LT01_AHH         := "LT003".LIM_Qb01,
        LT01_AH          := "LT003".LIM_Qb02,
        LT01_AL          := "LT003".LIM_Qb03,
        LT01_ALL         := "LT003".LIM_Qb04,
        LT01_ERR         := "LT003".QERR,
        XV_Bottom_OPN    := ,
        XV_Bottom_CLS    := ,
        XV_Bottom_MERR   := ,
        BV_Bottom_OPN    := "MV003".QOPEN,
        BV_Bottom_CLS    := "MV003".QCLOSE,
        BV_Bottom_MERR   := "MV003".QMON_ERR,
        BV_Tran_M04_OPN  := "MV003".QOPEN,
        BV_Tran_M04_CLS  := "MV003".QCLOSE,
        BV_Tran_M04_MERR := "MV003".QMON_ERR,
        steptime_s       := ,
        steptime_m       := ,
        steptime_h       := ,
        first_scan       := ,
        last_scan        := ,
        error_index_db   := ,
        Owner            := ,
        Status           := ,
        CM_error         := ,
        CM_error_no      := ,
        q_bACTVIE        := ,
        Level            := ,
        Pressure         := ,
        Pump_ON          := "M102".L_ON,
        Pump_AUT         := "M102".L_AUT,
        PIC01_EXT        := "LIC003".L_REMOTE,
        PIC01_SP         := "LIC003".HMI_SP_INT,
        PIC01_AUT        := "LIC003".L_AUT,
        PIC01_VAL_OUT    := "LIC003".HMI_MAN,
        PIC01_SET_SP     := "LIC003".Set_SP,
        PIC01_SET_OUT    := "LIC003".Set_Output,
        XV_Bottom_CMD    := ,
        BV_Bottom_CMD    := "MV003".AUT_OP,
        BV_Tran_M04_CMD  := "MV003".AUT_OP
      );
END_FUNCTION

FUNCTION "EM_Instance_4_fc" : Void   // FC1, STL
TITLE = _fc
{ S7_Optimized_Access := 'TRUE' }
VERSION : 0.1
// test
// stored: AutoNumber true, UDAEnableTagReadback false
BEGIN

NETWORK
TITLE = Main
// comment:


// Call the EM FB with the corresponding DB instance
      CALL  "EM_I_OUT", "EM_Instance_4"
      ( sampletime       := ,
        em_id            := 29,
        Request          := ,
        Command          := ,
        Pressure_SP      := ,
        Pump_RUN         := "M103".QNOFF2,
        Pump_QERR        := "M103".QERR,
        Pump_EERR        := "M103".QERR_EXT,
        FS01_PV          := "LS002".QON,
        PIC01_PV         := "LIC004".PV,
        PIC01_ERR        := "LIC004".QERR,
        LT01_PV          := "LT004".QfVal,
        LT01_AHH         := "LT004".LIM_Qb01,
        LT01_AH          := "LT004".LIM_Qb02,
        LT01_AL          := "LT004".LIM_Qb03,
        LT01_ALL         := "LT004".LIM_Qb04,
        LT01_ERR         := "LT004".QERR,
        XV_Bottom_OPN    := ,
        XV_Bottom_CLS    := ,
        XV_Bottom_MERR   := ,
        BV_Bottom_OPN    := "MV004".QOPEN,
        BV_Bottom_CLS    := "MV004".QCLOSE,
        BV_Bottom_MERR   := "MV004".QMON_ERR,
        BV_Tran_M04_OPN  := "MV003".QOPEN,
        BV_Tran_M04_CLS  := "MV003".QCLOSE,
        BV_Tran_M04_MERR := "MV003".QMON_ERR,
        steptime_s       := ,
        steptime_m       := ,
        steptime_h       := ,
        first_scan       := ,
        last_scan        := ,
        error_index_db   := ,
        Owner            := ,
        Status           := ,
        CM_error         := ,
        CM_error_no      := ,
        q_bACTVIE        := ,
        Level            := ,
        Pressure         := ,
        Pump_ON          := "M103".L_ON,
        Pump_AUT         := "M103".L_AUT,
        PIC01_EXT        := "LIC004".L_REMOTE,
        PIC01_SP         := "LIC004".HMI_SP_INT,
        PIC01_AUT        := "LIC004".L_AUT,
        PIC01_VAL_OUT    := "LIC004".HMI_MAN,
        PIC01_SET_SP     := "LIC004".Set_SP,
        PIC01_SET_OUT    := "LIC004".Set_Output,
        XV_Bottom_CMD    := ,
        BV_Bottom_CMD    := "MV004".AUT_OP,
        BV_Tran_M04_CMD  := "MV003".AUT_OP
      );
END_FUNCTION

FUNCTION "EM_Instance_5_fc" : Void   // FC1, STL
TITLE = _fc
{ S7_Optimized_Access := 'TRUE' }
VERSION : 0.1
// test
// stored: AutoNumber true, UDAEnableTagReadback false
BEGIN

NETWORK
TITLE = Main
// comment:


// Call the EM FB with the corresponding DB instance
      CALL  "EM_I_OUT", "EM_Instance_5"
      ( sampletime       := ,
        em_id            := 30,
        Request          := ,
        Command          := ,
        Pressure_SP      := ,
        Pump_RUN         := "M104".QNOFF2,
        Pump_QERR        := "M104".QERR,
        Pump_EERR        := "M104".QERR_EXT,
        FS01_PV          := "LS002".QON,
        PIC01_PV         := "LIC005".PV,
        PIC01_ERR        := "LIC005".QERR,
        LT01_PV          := "LT005".QfVal,
        LT01_AHH         := "LT005".LIM_Qb01,
        LT01_AH          := "LT005".LIM_Qb02,
        LT01_AL          := "LT005".LIM_Qb03,
        LT01_ALL         := "LT005".LIM_Qb04,
        LT01_ERR         := "LT005".QERR,
        XV_Bottom_OPN    := ,
        XV_Bottom_CLS    := ,
        XV_Bottom_MERR   := ,
        BV_Bottom_OPN    := "MV005".QOPEN,
        BV_Bottom_CLS    := "MV005".QCLOSE,
        BV_Bottom_MERR   := "MV005".QMON_ERR,
        BV_Tran_M04_OPN  := "MV003".QOPEN,
        BV_Tran_M04_CLS  := "MV003".QCLOSE,
        BV_Tran_M04_MERR := "MV003".QMON_ERR,
        steptime_s       := ,
        steptime_m       := ,
        steptime_h       := ,
        first_scan       := ,
        last_scan        := ,
        error_index_db   := ,
        Owner            := ,
        Status           := ,
        CM_error         := ,
        CM_error_no      := ,
        q_bACTVIE        := ,
        Level            := ,
        Pressure         := ,
        Pump_ON          := "M104".L_ON,
        Pump_AUT         := "M104".L_AUT,
        PIC01_EXT        := "LIC005".L_REMOTE,
        PIC01_SP         := "LIC005".HMI_SP_INT,
        PIC01_AUT        := "LIC005".L_AUT,
        PIC01_VAL_OUT    := "LIC005".HMI_MAN,
        PIC01_SET_SP     := "LIC005".Set_SP,
        PIC01_SET_OUT    := "LIC005".Set_Output,
        XV_Bottom_CMD    := ,
        BV_Bottom_CMD    := "MV005".AUT_OP,
        BV_Tran_M04_CMD  := "MV003".AUT_OP
      );
END_FUNCTION

FUNCTION "EM_Instance_6_fc" : Void   // FC1, STL
TITLE = _fc
{ S7_Optimized_Access := 'TRUE' }
VERSION : 0.1
// test
// stored: AutoNumber true, UDAEnableTagReadback false
BEGIN

NETWORK
TITLE = Main
// comment:


// Call the EM FB with the corresponding DB instance
      CALL  "EM_I_OUT", "EM_Instance_6"
      ( sampletime       := ,
        em_id            := 31,
        Request          := ,
        Command          := ,
        Pressure_SP      := ,
        Pump_RUN         := "M105".QNOFF2,
        Pump_QERR        := "M105".QERR,
        Pump_EERR        := "M105".QERR_EXT,
        FS01_PV          := "LS002".QON,
        PIC01_PV         := "LIC006".PV,
        PIC01_ERR        := "LIC006".QERR,
        LT01_PV          := "LT006".QfVal,
        LT01_AHH         := "LT006".LIM_Qb01,
        LT01_AH          := "LT006".LIM_Qb02,
        LT01_AL          := "LT006".LIM_Qb03,
        LT01_ALL         := "LT006".LIM_Qb04,
        LT01_ERR         := "LT006".QERR,
        XV_Bottom_OPN    := ,
        XV_Bottom_CLS    := ,
        XV_Bottom_MERR   := ,
        BV_Bottom_OPN    := "MV006".QOPEN,
        BV_Bottom_CLS    := "MV006".QCLOSE,
        BV_Bottom_MERR   := "MV006".QMON_ERR,
        BV_Tran_M04_OPN  := "MV003".QOPEN,
        BV_Tran_M04_CLS  := "MV003".QCLOSE,
        BV_Tran_M04_MERR := "MV003".QMON_ERR,
        steptime_s       := ,
        steptime_m       := ,
        steptime_h       := ,
        first_scan       := ,
        last_scan        := ,
        error_index_db   := ,
        Owner            := ,
        Status           := ,
        CM_error         := ,
        CM_error_no      := ,
        q_bACTVIE        := ,
        Level            := ,
        Pressure         := ,
        Pump_ON          := "M105".L_ON,
        Pump_AUT         := "M105".L_AUT,
        PIC01_EXT        := "LIC006".L_REMOTE,
        PIC01_SP         := "LIC006".HMI_SP_INT,
        PIC01_AUT        := "LIC006".L_AUT,
        PIC01_VAL_OUT    := "LIC006".HMI_MAN,
        PIC01_SET_SP     := "LIC006".Set_SP,
        PIC01_SET_OUT    := "LIC006".Set_Output,
        XV_Bottom_CMD    := ,
        BV_Bottom_CMD    := "MV006".AUT_OP,
        BV_Tran_M04_CMD  := "MV003".AUT_OP
      );
END_FUNCTION

FUNCTION "EM_Instance_7_fc" : Void   // FC1, STL
TITLE = _fc
{ S7_Optimized_Access := 'TRUE' }
VERSION : 0.1
// test
// stored: AutoNumber true, UDAEnableTagReadback false
BEGIN

NETWORK
TITLE = Main
// comment:


// Call the EM FB with the corresponding DB instance
      CALL  "EM_I_OUT", "EM_Instance_7"
      ( sampletime       := ,
        em_id            := 32,
        Request          := ,
        Command          := ,
        Pressure_SP      := ,
        Pump_RUN         := "M106".QNOFF2,
        Pump_QERR        := "M106".QERR,
        Pump_EERR        := "M106".QERR_EXT,
        FS01_PV          := "LS002".QON,
        PIC01_PV         := "FIC100".PV,
        PIC01_ERR        := "FIC100".QERR,
        LT01_PV          := "LT007".QfVal,
        LT01_AHH         := "LT007".LIM_Qb01,
        LT01_AH          := "LT007".LIM_Qb02,
        LT01_AL          := "LT007".LIM_Qb03,
        LT01_ALL         := "LT007".LIM_Qb04,
        LT01_ERR         := "LT007".QERR,
        XV_Bottom_OPN    := ,
        XV_Bottom_CLS    := ,
        XV_Bottom_MERR   := ,
        BV_Bottom_OPN    := "MV007".QOPEN,
        BV_Bottom_CLS    := "MV007".QCLOSE,
        BV_Bottom_MERR   := "MV007".QMON_ERR,
        BV_Tran_M04_OPN  := "MV003".QOPEN,
        BV_Tran_M04_CLS  := "MV003".QCLOSE,
        BV_Tran_M04_MERR := "MV003".QMON_ERR,
        steptime_s       := ,
        steptime_m       := ,
        steptime_h       := ,
        first_scan       := ,
        last_scan        := ,
        error_index_db   := ,
        Owner            := ,
        Status           := ,
        CM_error         := ,
        CM_error_no      := ,
        q_bACTVIE        := ,
        Level            := ,
        Pressure         := ,
        Pump_ON          := "M106".L_ON,
        Pump_AUT         := "M106".L_AUT,
        PIC01_EXT        := "FIC100".L_REMOTE,
        PIC01_SP         := "FIC100".HMI_SP_INT,
        PIC01_AUT        := "FIC100".L_AUT,
        PIC01_VAL_OUT    := "FIC100".HMI_MAN,
        PIC01_SET_SP     := "FIC100".Set_SP,
        PIC01_SET_OUT    := "FIC100".Set_Output,
        XV_Bottom_CMD    := ,
        BV_Bottom_CMD    := "MV007".AUT_OP,
        BV_Tran_M04_CMD  := "MV003".AUT_OP
      );
END_FUNCTION

FUNCTION "EM_Instance_8_fc" : Void   // FC1, STL
TITLE = _fc
{ S7_Optimized_Access := 'TRUE' }
VERSION : 0.1
// test
// stored: AutoNumber true, UDAEnableTagReadback false
BEGIN

NETWORK
TITLE = Main
// comment:


// Call the EM FB with the corresponding DB instance
      CALL  "EM_I_OUT", "EM_Instance_8"
      ( sampletime       := ,
        em_id            := 33,
        Request          := ,
        Command          := ,
        Pressure_SP      := ,
        Pump_RUN         := "M106".QNOFF2,
        Pump_QERR        := "M106".QERR,
        Pump_EERR        := "M106".QERR_EXT,
        FS01_PV          := "LS002".QON,
        PIC01_PV         := "FIC101".PV,
        PIC01_ERR        := "FIC101".QERR,
        LT01_PV          := "LT100".QfVal,
        LT01_AHH         := "LT100".LIM_Qb01,
        LT01_AH          := "LT100".LIM_Qb02,
        LT01_AL          := "LT100".LIM_Qb03,
        LT01_ALL         := "LT100".LIM_Qb04,
        LT01_ERR         := "LT100".QERR,
        XV_Bottom_OPN    := ,
        XV_Bottom_CLS    := ,
        XV_Bottom_MERR   := ,
        BV_Bottom_OPN    := "MV007".QOPEN,
        BV_Bottom_CLS    := "MV007".QCLOSE,
        BV_Bottom_MERR   := "MV007".QMON_ERR,
        BV_Tran_M04_OPN  := "MV003".QOPEN,
        BV_Tran_M04_CLS  := "MV003".QCLOSE,
        BV_Tran_M04_MERR := "MV003".QMON_ERR,
        steptime_s       := ,
        steptime_m       := ,
        steptime_h       := ,
        first_scan       := ,
        last_scan        := ,
        error_index_db   := ,
        Owner            := ,
        Status           := ,
        CM_error         := ,
        CM_error_no      := ,
        q_bACTVIE        := ,
        Level            := ,
        Pressure         := ,
        Pump_ON          := "M106".L_ON,
        Pump_AUT         := "M106".L_AUT,
        PIC01_EXT        := "FIC101".L_REMOTE,
        PIC01_SP         := "FIC101".HMI_SP_INT,
        PIC01_AUT        := "FIC101".L_AUT,
        PIC01_VAL_OUT    := "FIC101".HMI_MAN,
        PIC01_SET_SP     := "FIC101".Set_SP,
        PIC01_SET_OUT    := "FIC101".Set_Output,
        XV_Bottom_CMD    := ,
        BV_Bottom_CMD    := "MV007".AUT_OP,
        BV_Tran_M04_CMD  := "MV003".AUT_OP
      );
END_FUNCTION

FUNCTION "EM_Instance_9_fc" : Void   // FC1, STL
TITLE = _fc
{ S7_Optimized_Access := 'TRUE' }
VERSION : 0.1
// test
// stored: AutoNumber true, UDAEnableTagReadback false
BEGIN

NETWORK
TITLE = Main
// comment:


// Call the EM FB with the corresponding DB instance
      CALL  "EM_I_OUT", "EM_Instance_9"
      ( sampletime       := ,
        em_id            := 34,
        Request          := ,
        Command          := ,
        Pressure_SP      := ,
        Pump_RUN         := "M106".QNOFF2,
        Pump_QERR        := "M106".QERR,
        Pump_EERR        := "M106".QERR_EXT,
        FS01_PV          := "LS002".QON,
        PIC01_PV         := "FIC101".PV,
        PIC01_ERR        := "FIC101".QERR,
        LT01_PV          := "LT200".QfVal,
        LT01_AHH         := "LT200".LIM_Qb01,
        LT01_AH          := "LT200".LIM_Qb02,
        LT01_AL          := "LT200".LIM_Qb03,
        LT01_ALL         := "LT200".LIM_Qb04,
        LT01_ERR         := "LT200".QERR,
        XV_Bottom_OPN    := ,
        XV_Bottom_CLS    := ,
        XV_Bottom_MERR   := ,
        BV_Bottom_OPN    := "MV007".QOPEN,
        BV_Bottom_CLS    := "MV007".QCLOSE,
        BV_Bottom_MERR   := "MV007".QMON_ERR,
        BV_Tran_M04_OPN  := "MV003".QOPEN,
        BV_Tran_M04_CLS  := "MV003".QCLOSE,
        BV_Tran_M04_MERR := "MV003".QMON_ERR,
        steptime_s       := ,
        steptime_m       := ,
        steptime_h       := ,
        first_scan       := ,
        last_scan        := ,
        error_index_db   := ,
        Owner            := ,
        Status           := ,
        CM_error         := ,
        CM_error_no      := ,
        q_bACTVIE        := ,
        Level            := ,
        Pressure         := ,
        Pump_ON          := "M106".L_ON,
        Pump_AUT         := "M106".L_AUT,
        PIC01_EXT        := "FIC101".L_REMOTE,
        PIC01_SP         := "FIC101".HMI_SP_INT,
        PIC01_AUT        := "FIC101".L_AUT,
        PIC01_VAL_OUT    := "FIC101".HMI_MAN,
        PIC01_SET_SP     := "FIC101".Set_SP,
        PIC01_SET_OUT    := "FIC101".Set_Output,
        XV_Bottom_CMD    := ,
        BV_Bottom_CMD    := "MV007".AUT_OP,
        BV_Tran_M04_CMD  := "MV003".AUT_OP
      );
END_FUNCTION

FUNCTION "FIC100_fc" : Void   // FC1, STL
TITLE = FIC100_fc
{ S7_Optimized_Access := 'TRUE' }
VERSION : 0.1
// test
// stored: AutoNumber true, UDAEnableTagReadback false
BEGIN

NETWORK
TITLE = Change PID Setpoints
// The phase FBs write on the operator setpoints of the PID-controller
// To avoid that the setpoints are always overwritten (and blocking operator control)
// we use pulses generated by the phase to set the setpoints only at specific moments
// i_fOCmdSP (setpoint)
// i_fOCmdMANOP (output)
      CALL  "BST_PIDAIN_400", "DB";


//Write the Operator_Setpoint
      A     "FIC100_sp".Set_SP;
      JCN   J001;

      L     "FIC100_sp".Operator_Setpoint;
      T     "FIC100".i_fOCmdSP;

J001: NOP   0;


//Write the Output_Value
      A     "FIC100_sp".Set_Output;
      JCN   J002;

      L     "FIC100_sp".Output_Value;
      T     "FIC100".i_fOCmdMANOP;

J002: NOP   0;



NETWORK
TITLE = Main
// comment: PLC1


//Call the CM FB with the corresponding DB instance
END_FUNCTION

FUNCTION_BLOCK "BST_PIDAIN_400"   // FB25, STL
{ S7_Optimized_Access := 'FALSE' }
VERSION : 0.1
// stored: AutoNumber false, CodeModifiedDate 2018-05-30T14:05:05.4814636Z, CompileDate 2018-05-30T14:05:05.4814635Z, CreationDate 2018-05-30T13:57:54.5148136Z, InterfaceModifiedDate 2018-05-30T14:05:02.6553018Z, IsConsistent true, IsKnowHowProtected false, ISMultiInstanceCapable true, IsWriteProtected false, LibraryConformanceStatus The object is library-conformant., ModifiedDate 2018-05-30T14:05:05.4814636Z, ParameterModified 2018-05-30T14:05:02.6553018Z, StructureModified 2018-05-30T14:05:02.6553018Z, UDAEnableTagReadback false
   VAR_INPUT
      L_REMOTE : Bool;
      HMI_SP_INT : Real;
      L_AUT : Bool;
      HMI_MAN : Real;
      PV : Real;
      Set_SP : Bool;
      Set_Output : Bool;
      i_fOCmdSP : Real;
      i_fOCmdMANOP : Real;
   END_VAR
   VAR_OUTPUT
      PV_OUT : Real;
      QERR : Bool;
      LMN : Real;
   END_VAR
BEGIN
END_FUNCTION_BLOCK

FUNCTION "FIC101_fc" : Void   // FC1, STL
TITLE = FIC101_fc
{ S7_Optimized_Access := 'TRUE' }
VERSION : 0.1
// test
// stored: AutoNumber true, UDAEnableTagReadback false
BEGIN

NETWORK
TITLE = Change PID Setpoints
// The phase FBs write on the operator setpoints of the PID-controller
// To avoid that the setpoints are always overwritten (and blocking operator control)
// we use pulses generated by the phase to set the setpoints only at specific moments
// i_fOCmdSP (setpoint)
// i_fOCmdMANOP (output)
      CALL  "BST_PIDAIN_400", "DB";


//Write the Operator_Setpoint
      A     "FIC101_sp".Set_SP;
      JCN   J001;

      L     "FIC101_sp".Operator_Setpoint;
      T     "FIC101".i_fOCmdSP;

J001: NOP   0;


//Write the Output_Value
      A     "FIC101_sp".Set_Output;
      JCN   J002;

      L     "FIC101_sp".Output_Value;
      T     "FIC101".i_fOCmdMANOP;

J002: NOP   0;



NETWORK
TITLE = Main
// comment: PLC1


//Call the CM FB with the corresponding DB instance
END_FUNCTION

FUNCTION "LIC001_fc" : Void   // FC1, STL
TITLE = LIC001_fc
{ S7_Optimized_Access := 'TRUE' }
VERSION : 0.1
// test
// stored: AutoNumber true, UDAEnableTagReadback false
BEGIN

NETWORK
TITLE = Change PID Setpoints
// The phase FBs write on the operator setpoints of the PID-controller
// To avoid that the setpoints are always overwritten (and blocking operator control)
// we use pulses generated by the phase to set the setpoints only at specific moments
// i_fOCmdSP (setpoint)
// i_fOCmdMANOP (output)
      CALL  "BST_DIGITAL_400", "DB";


//Write the Operator_Setpoint
      A     "LIC001_sp".Set_SP;
      JCN   J001;

      L     "LIC001_sp".Operator_Setpoint;
      T     "LIC001".i_fOCmdSP;

J001: NOP   0;


//Write the Output_Value
      A     "LIC001_sp".Set_Output;
      JCN   J002;

      L     "LIC001_sp".Output_Value;
      T     "LIC001".i_fOCmdMANOP;

J002: NOP   0;



NETWORK
TITLE = Main
// comment: PLC1


//Call the CM FB with the corresponding DB instance
END_FUNCTION

FUNCTION_BLOCK "BST_DIGITAL_400"   // FB24, STL
{ S7_Optimized_Access := 'FALSE' }
VERSION : 0.1
// stored: AutoNumber false, CodeModifiedDate 2018-05-30T14:06:41.0879319Z, CompileDate 2018-05-30T14:06:41.0879318Z, CreationDate 2018-05-30T13:57:30.9234642Z, InterfaceModifiedDate 2018-05-30T14:02:05.4231647Z, IsConsistent true, IsKnowHowProtected false, ISMultiInstanceCapable true, IsWriteProtected false, LibraryConformanceStatus The object is library-conformant., ModifiedDate 2018-05-30T14:06:41.0879319Z, ParameterModified 2018-05-30T14:02:05.4231647Z, StructureModified 2018-05-30T14:02:05.4231647Z, UDAEnableTagReadback false
   VAR_INPUT
      i_bInp : Bool;
   END_VAR
   VAR_OUTPUT
      QON : Bool;
   END_VAR
BEGIN
END_FUNCTION_BLOCK

FUNCTION "LIC002_fc" : Void   // FC1, STL
TITLE = LIC002_fc
{ S7_Optimized_Access := 'TRUE' }
VERSION : 0.1
// test
// stored: AutoNumber true, UDAEnableTagReadback false
BEGIN

NETWORK
TITLE = Change PID Setpoints
// The phase FBs write on the operator setpoints of the PID-controller
// To avoid that the setpoints are always overwritten (and blocking operator control)
// we use pulses generated by the phase to set the setpoints only at specific moments
// i_fOCmdSP (setpoint)
// i_fOCmdMANOP (output)
      CALL  "BST_PIDAIN_400", "DB";


//Write the Operator_Setpoint
      A     "LIC002_sp".Set_SP;
      JCN   J001;

      L     "LIC002_sp".Operator_Setpoint;
      T     "LIC002".i_fOCmdSP;

J001: NOP   0;


//Write the Output_Value
      A     "LIC002_sp".Set_Output;
      JCN   J002;

      L     "LIC002_sp".Output_Value;
      T     "LIC002".i_fOCmdMANOP;

J002: NOP   0;



NETWORK
TITLE = Main
// comment: PLC1


//Call the CM FB with the corresponding DB instance
END_FUNCTION

FUNCTION "LIC003_fc" : Void   // FC1, STL
TITLE = LIC003_fc
{ S7_Optimized_Access := 'TRUE' }
VERSION : 0.1
// test
// stored: AutoNumber true, UDAEnableTagReadback false
BEGIN

NETWORK
TITLE = Change PID Setpoints
// The phase FBs write on the operator setpoints of the PID-controller
// To avoid that the setpoints are always overwritten (and blocking operator control)
// we use pulses generated by the phase to set the setpoints only at specific moments
// i_fOCmdSP (setpoint)
// i_fOCmdMANOP (output)
      CALL  "BST_PIDAIN_400", "DB";


//Write the Operator_Setpoint
      A     "LIC003_sp".Set_SP;
      JCN   J001;

      L     "LIC003_sp".Operator_Setpoint;
      T     "LIC003".i_fOCmdSP;

J001: NOP   0;


//Write the Output_Value
      A     "LIC003_sp".Set_Output;
      JCN   J002;

      L     "LIC003_sp".Output_Value;
      T     "LIC003".i_fOCmdMANOP;

J002: NOP   0;



NETWORK
TITLE = Main
// comment: PLC1


//Call the CM FB with the corresponding DB instance
END_FUNCTION

FUNCTION "LIC004_fc" : Void   // FC1, STL
TITLE = LIC004_fc
{ S7_Optimized_Access := 'TRUE' }
VERSION : 0.1
// test
// stored: AutoNumber true, UDAEnableTagReadback false
BEGIN

NETWORK
TITLE = Change PID Setpoints
// The phase FBs write on the operator setpoints of the PID-controller
// To avoid that the setpoints are always overwritten (and blocking operator control)
// we use pulses generated by the phase to set the setpoints only at specific moments
// i_fOCmdSP (setpoint)
// i_fOCmdMANOP (output)
      CALL  "BST_PIDAIN_400", "DB";


//Write the Operator_Setpoint
      A     "LIC004_sp".Set_SP;
      JCN   J001;

      L     "LIC004_sp".Operator_Setpoint;
      T     "LIC004".i_fOCmdSP;

J001: NOP   0;


//Write the Output_Value
      A     "LIC004_sp".Set_Output;
      JCN   J002;

      L     "LIC004_sp".Output_Value;
      T     "LIC004".i_fOCmdMANOP;

J002: NOP   0;



NETWORK
TITLE = Main
// comment: PLC1


//Call the CM FB with the corresponding DB instance
END_FUNCTION

FUNCTION "LIC005_fc" : Void   // FC1, STL
TITLE = LIC005_fc
{ S7_Optimized_Access := 'TRUE' }
VERSION : 0.1
// test
// stored: AutoNumber true, UDAEnableTagReadback false
BEGIN

NETWORK
TITLE = Change PID Setpoints
// The phase FBs write on the operator setpoints of the PID-controller
// To avoid that the setpoints are always overwritten (and blocking operator control)
// we use pulses generated by the phase to set the setpoints only at specific moments
// i_fOCmdSP (setpoint)
// i_fOCmdMANOP (output)
      CALL  "BST_PIDAIN_400", "DB";


//Write the Operator_Setpoint
      A     "LIC005_sp".Set_SP;
      JCN   J001;

      L     "LIC005_sp".Operator_Setpoint;
      T     "LIC005".i_fOCmdSP;

J001: NOP   0;


//Write the Output_Value
      A     "LIC005_sp".Set_Output;
      JCN   J002;

      L     "LIC005_sp".Output_Value;
      T     "LIC005".i_fOCmdMANOP;

J002: NOP   0;



NETWORK
TITLE = Main
// comment: PLC1


//Call the CM FB with the corresponding DB instance
END_FUNCTION

FUNCTION "LIC006_fc" : Void   // FC1, STL
TITLE = LIC006_fc
{ S7_Optimized_Access := 'TRUE' }
VERSION : 0.1
// test
// stored: AutoNumber true, UDAEnableTagReadback false
BEGIN

NETWORK
TITLE = Change PID Setpoints
// The phase FBs write on the operator setpoints of the PID-controller
// To avoid that the setpoints are always overwritten (and blocking operator control)
// we use pulses generated by the phase to set the setpoints only at specific moments
// i_fOCmdSP (setpoint)
// i_fOCmdMANOP (output)
      CALL  "BST_PIDAIN_400", "DB";


//Write the Operator_Setpoint
      A     "LIC006_sp".Set_SP;
      JCN   J001;

      L     "LIC006_sp".Operator_Setpoint;
      T     "LIC006".i_fOCmdSP;

J001: NOP   0;


//Write the Output_Value
      A     "LIC006_sp".Set_Output;
      JCN   J002;

      L     "LIC006_sp".Output_Value;
      T     "LIC006".i_fOCmdMANOP;

J002: NOP   0;



NETWORK
TITLE = Main
// comment: PLC1


//Call the CM FB with the corresponding DB instance
END_FUNCTION

FUNCTION "LS001_fc" : Void   // FC1, STL
TITLE = LS001_fc
{ S7_Optimized_Access := 'TRUE' }
VERSION : 0.1
// test
// stored: AutoNumber true, UDAEnableTagReadback false
BEGIN

NETWORK
TITLE = Main
// comment: PLC1
      CALL  "BST_ANALOG_400", "DB";


//Call the CM FB with the corresponding DB instance
END_FUNCTION

FUNCTION_BLOCK "BST_ANALOG_400"   // FB23, STL
{ S7_Optimized_Access := 'FALSE' }
VERSION : 0.1
// stored: AutoNumber false, CodeModifiedDate 2018-05-30T14:01:37.8315867Z, CompileDate 2018-05-30T14:01:37.8315866Z, CreationDate 2018-05-30T13:57:04.4029473Z, InterfaceModifiedDate 2018-05-30T14:01:33.7723544Z, IsConsistent true, IsKnowHowProtected false, ISMultiInstanceCapable true, IsWriteProtected false, LibraryConformanceStatus The object is library-conformant., ModifiedDate 2018-05-30T14:01:37.8315867Z, ParameterModified 2018-05-30T14:01:33.7723544Z, StructureModified 2018-05-30T14:01:33.7723544Z, UDAEnableTagReadback false
   VAR_INPUT
      wVal : Real;
   END_VAR
   VAR_OUTPUT
      QfVal : Real;
      LIM_Qb01 : Bool;
      LIM_Qb02 : Bool;
      LIM_Qb03 : Bool;
      LIM_b04 : Bool;
      QERR : Bool;
   END_VAR
BEGIN
END_FUNCTION_BLOCK

FUNCTION "LS002_fc" : Void   // FC1, STL
TITLE = LS002_fc
{ S7_Optimized_Access := 'TRUE' }
VERSION : 0.1
// test
// stored: AutoNumber true, UDAEnableTagReadback false
BEGIN

NETWORK
TITLE = Main
// comment: PLC1
      CALL  "BST_DIGITAL_400", "DB";


//Call the CM FB with the corresponding DB instance
END_FUNCTION

FUNCTION "LT001_fc" : Void   // FC1, STL
TITLE = LT001_fc
{ S7_Optimized_Access := 'TRUE' }
VERSION : 0.1
// test
// stored: AutoNumber true, UDAEnableTagReadback false
BEGIN

NETWORK
TITLE = Main
// comment: PLC1
      CALL  "BST_SINAG120_400", "DB";


//Call the CM FB with the corresponding DB instance
END_FUNCTION

FUNCTION_BLOCK "BST_SINAG120_400"   // FB22, STL
{ S7_Optimized_Access := 'FALSE' }
VERSION : 0.1
// stored: AutoNumber false, CodeModifiedDate 2018-05-30T14:00:08.4304732Z, CompileDate 2018-05-30T14:00:08.4304731Z, CreationDate 2018-05-30T13:56:31.6980767Z, InterfaceModifiedDate 2018-05-30T13:59:44.6951155Z, IsConsistent true, IsKnowHowProtected false, ISMultiInstanceCapable true, IsWriteProtected false, LibraryConformanceStatus The object is library-conformant., ModifiedDate 2018-05-30T14:00:08.4304732Z, ParameterModified 2018-05-30T13:59:44.6951155Z, StructureModified 2018-05-30T13:59:44.6951155Z, UDAEnableTagReadback false
   VAR_INPUT
      L_ON : Bool;
      L_AUT : Bool;
   END_VAR
   VAR_OUTPUT
      QNOFF2 : Bool;
      QERR : Bool;
      QERR_EXT : Bool;
   END_VAR
BEGIN
END_FUNCTION_BLOCK

FUNCTION "LT002_fc" : Void   // FC1, STL
TITLE = LT002_fc
{ S7_Optimized_Access := 'TRUE' }
VERSION : 0.1
// test
// stored: AutoNumber true, UDAEnableTagReadback false
BEGIN

NETWORK
TITLE = Main
// comment: PLC1
      CALL  "BST_ANALOG_400", "DB";


//Call the CM FB with the corresponding DB instance
END_FUNCTION

FUNCTION "LT003_fc" : Void   // FC1, STL
TITLE = LT003_fc
{ S7_Optimized_Access := 'TRUE' }
VERSION : 0.1
// test
// stored: AutoNumber true, UDAEnableTagReadback false
BEGIN

NETWORK
TITLE = Main
// comment: PLC1
      CALL  "BST_ANALOG_400", "DB";


//Call the CM FB with the corresponding DB instance
END_FUNCTION

FUNCTION "LT004_fc" : Void   // FC1, STL
TITLE = LT004_fc
{ S7_Optimized_Access := 'TRUE' }
VERSION : 0.1
// test
// stored: AutoNumber true, UDAEnableTagReadback false
BEGIN

NETWORK
TITLE = Main
// comment: PLC1
      CALL  "BST_ANALOG_400", "DB";


//Call the CM FB with the corresponding DB instance
END_FUNCTION

FUNCTION "LT005_fc" : Void   // FC1, STL
TITLE = LT005_fc
{ S7_Optimized_Access := 'TRUE' }
VERSION : 0.1
// test
// stored: AutoNumber true, UDAEnableTagReadback false
BEGIN

NETWORK
TITLE = Main
// comment: PLC1
      CALL  "BST_ANALOG_400", "DB";


//Call the CM FB with the corresponding DB instance
END_FUNCTION

FUNCTION "LT006_fc" : Void   // FC1, STL
TITLE = LT006_fc
{ S7_Optimized_Access := 'TRUE' }
VERSION : 0.1
// test
// stored: AutoNumber true, UDAEnableTagReadback false
BEGIN

NETWORK
TITLE = Main
// comment: PLC1
      CALL  "BST_ANALOG_400", "DB";


//Call the CM FB with the corresponding DB instance
END_FUNCTION

FUNCTION "LT007_fc" : Void   // FC1, STL
TITLE = LT007_fc
{ S7_Optimized_Access := 'TRUE' }
VERSION : 0.1
// test
// stored: AutoNumber true, UDAEnableTagReadback false
BEGIN

NETWORK
TITLE = Main
// comment: PLC1
      CALL  "BST_ANALOG_400", "DB";


//Call the CM FB with the corresponding DB instance
END_FUNCTION

FUNCTION "LT100_fc" : Void   // FC1, STL
TITLE = LT100_fc
{ S7_Optimized_Access := 'TRUE' }
VERSION : 0.1
// test
// stored: AutoNumber true, UDAEnableTagReadback false
BEGIN

NETWORK
TITLE = Main
// comment: PLC1
      CALL  "BST_ANALOG_400", "DB";


//Call the CM FB with the corresponding DB instance
END_FUNCTION

FUNCTION "LT101_fc" : Void   // FC1, STL
TITLE = LT101_fc
{ S7_Optimized_Access := 'TRUE' }
VERSION : 0.1
// test
// stored: AutoNumber true, UDAEnableTagReadback false
BEGIN

NETWORK
TITLE = Main
// comment: PLC1
      CALL  "BST_ANALOG_400", "DB";


//Call the CM FB with the corresponding DB instance
END_FUNCTION

FUNCTION "LT200_fc" : Void   // FC1, STL
TITLE = LT200_fc
{ S7_Optimized_Access := 'TRUE' }
VERSION : 0.1
// test
// stored: AutoNumber true, UDAEnableTagReadback false
BEGIN

NETWORK
TITLE = Main
// comment: PLC1
      CALL  "BST_ANALOG_400", "DB";


//Call the CM FB with the corresponding DB instance
END_FUNCTION

FUNCTION "LT201_fc" : Void   // FC1, STL
TITLE = LT201_fc
{ S7_Optimized_Access := 'TRUE' }
VERSION : 0.1
// test
// stored: AutoNumber true, UDAEnableTagReadback false
BEGIN

NETWORK
TITLE = Main
// comment: PLC1
      CALL  "BST_ANALOG_400", "DB";


//Call the CM FB with the corresponding DB instance
END_FUNCTION

FUNCTION "M100_fc" : Void   // FC1, STL
TITLE = M100_fc
{ S7_Optimized_Access := 'TRUE' }
VERSION : 0.1
// test
// stored: AutoNumber true, UDAEnableTagReadback false
BEGIN

NETWORK
TITLE = Main
// comment: PLC1
      CALL  "BST_MOTOR_400", "DB";


//Call the CM FB with the corresponding DB instance
END_FUNCTION

FUNCTION_BLOCK "BST_MOTOR_400"   // FB21, STL
{ S7_Optimized_Access := 'FALSE' }
VERSION : 0.1
// stored: AutoNumber false, CodeModifiedDate 2018-05-30T13:59:14.5053889Z, CompileDate 2018-05-30T13:59:14.5053888Z, CreationDate 2018-05-30T13:55:26.8283664Z, InterfaceModifiedDate 2018-05-30T13:59:03.2547453Z, IsConsistent true, IsKnowHowProtected false, ISMultiInstanceCapable true, IsWriteProtected false, LibraryConformanceStatus The object is library-conformant., ModifiedDate 2018-05-30T13:59:14.5053889Z, ParameterModified 2018-05-30T13:59:03.2547453Z, StructureModified 2018-05-30T13:59:03.2547453Z, UDAEnableTagReadback false
   VAR_INPUT
      AUTO_ON : Bool;
      L_AUT : Bool;
      FB_ON : Bool;
      ERR_EXTERN : Bool;
   END_VAR
   VAR_OUTPUT
      QRUN : Bool;
      QSTOP : Bool;
      QCMD_ON : Bool;
      QMON_ERR : Bool;
      QMPS : Bool;
      QERR : Bool;
   END_VAR
BEGIN
END_FUNCTION_BLOCK

FUNCTION "M101_fc" : Void   // FC1, STL
TITLE = M101_fc
{ S7_Optimized_Access := 'TRUE' }
VERSION : 0.1
// test
// stored: AutoNumber true, UDAEnableTagReadback false
BEGIN

NETWORK
TITLE = Main
// comment: PLC1
      CALL  "BST_SINAG120_400", "DB";


//Call the CM FB with the corresponding DB instance
END_FUNCTION

FUNCTION "M102_fc" : Void   // FC1, STL
TITLE = M102_fc
{ S7_Optimized_Access := 'TRUE' }
VERSION : 0.1
// test
// stored: AutoNumber true, UDAEnableTagReadback false
BEGIN

NETWORK
TITLE = Main
// comment: PLC1
      CALL  "BST_SINAG120_400", "DB";


//Call the CM FB with the corresponding DB instance
END_FUNCTION

FUNCTION "M103_fc" : Void   // FC1, STL
TITLE = M103_fc
{ S7_Optimized_Access := 'TRUE' }
VERSION : 0.1
// test
// stored: AutoNumber true, UDAEnableTagReadback false
BEGIN

NETWORK
TITLE = Main
// comment: PLC1
      CALL  "BST_SINAG120_400", "DB";


//Call the CM FB with the corresponding DB instance
END_FUNCTION

FUNCTION "M104_fc" : Void   // FC1, STL
TITLE = M104_fc
{ S7_Optimized_Access := 'TRUE' }
VERSION : 0.1
// test
// stored: AutoNumber true, UDAEnableTagReadback false
BEGIN

NETWORK
TITLE = Main
// comment: PLC1
      CALL  "BST_SINAG120_400", "DB";


//Call the CM FB with the corresponding DB instance
END_FUNCTION

FUNCTION "M105_fc" : Void   // FC1, STL
TITLE = M105_fc
{ S7_Optimized_Access := 'TRUE' }
VERSION : 0.1
// test
// stored: AutoNumber true, UDAEnableTagReadback false
BEGIN

NETWORK
TITLE = Main
// comment: PLC1
      CALL  "BST_SINAG120_400", "DB";


//Call the CM FB with the corresponding DB instance
END_FUNCTION

FUNCTION "M106_fc" : Void   // FC1, STL
TITLE = M106_fc
{ S7_Optimized_Access := 'TRUE' }
VERSION : 0.1
// test
// stored: AutoNumber true, UDAEnableTagReadback false
BEGIN

NETWORK
TITLE = Main
// comment: PLC1
      CALL  "BST_SINAG120_400", "DB";


//Call the CM FB with the corresponding DB instance
END_FUNCTION

FUNCTION "MV001_fc" : Void   // FC1, STL
TITLE = MV001_fc
{ S7_Optimized_Access := 'TRUE' }
VERSION : 0.1
// test
// stored: AutoNumber true, UDAEnableTagReadback false
BEGIN

NETWORK
TITLE = Main
// comment: PLC1
      CALL  "BST_VALVE_400", "DB";


//Call the CM FB with the corresponding DB instance
END_FUNCTION

FUNCTION_BLOCK "BST_VALVE_400"   // FB20, STL
{ S7_Optimized_Access := 'FALSE' }
VERSION : 0.1
// stored: AutoNumber false, CodeModifiedDate 2018-05-30T13:28:59.5225777Z, CompileDate 2018-05-30T13:28:59.5215776Z, CreationDate 2018-05-30T13:22:11.3692328Z, InterfaceModifiedDate 2018-05-30T13:23:22.3522927Z, IsConsistent true, IsKnowHowProtected false, ISMultiInstanceCapable true, IsWriteProtected false, LibraryConformanceStatus The object is library-conformant., ModifiedDate 2018-05-30T13:28:59.5225777Z, ParameterModified 2018-05-30T13:23:22.3522927Z, StructureModified 2018-05-30T13:23:22.3522927Z, UDAEnableTagReadback false
   VAR_INPUT
      AUT_OP : Bool;   // Auto command from program
      FB_OPEN : Bool;   // Feedback Open
      FB_CLOSE : Bool;   // Feedback Close
   END_VAR
   VAR_OUTPUT
      QOPEN : Bool;   // Opened
      QCLOSE : Bool;   // Closed
      QMON_ERR : Bool;   // Monitoring Error
      QCMD_OP : Bool;   // Command to Valve
   END_VAR
BEGIN
END_FUNCTION_BLOCK

FUNCTION "MV002_fc" : Void   // FC1, STL
TITLE = MV002_fc
{ S7_Optimized_Access := 'TRUE' }
VERSION : 0.1
// test
// stored: AutoNumber true, UDAEnableTagReadback false
BEGIN

NETWORK
TITLE = Main
// comment: PLC1
      CALL  "BST_VALVE_400", "DB";


//Call the CM FB with the corresponding DB instance
END_FUNCTION

FUNCTION "MV003_fc" : Void   // FC1, STL
TITLE = MV003_fc
{ S7_Optimized_Access := 'TRUE' }
VERSION : 0.1
// test
// stored: AutoNumber true, UDAEnableTagReadback false
BEGIN

NETWORK
TITLE = Main
// comment: PLC1
      CALL  "BST_VALVE_400", "DB";


//Call the CM FB with the corresponding DB instance
END_FUNCTION

FUNCTION "MV004_fc" : Void   // FC1, STL
TITLE = MV004_fc
{ S7_Optimized_Access := 'TRUE' }
VERSION : 0.1
// test
// stored: AutoNumber true, UDAEnableTagReadback false
BEGIN

NETWORK
TITLE = Main
// comment: PLC1
      CALL  "BST_VALVE_400", "DB";


//Call the CM FB with the corresponding DB instance
END_FUNCTION

FUNCTION "MV005_fc" : Void   // FC1, STL
TITLE = MV005_fc
{ S7_Optimized_Access := 'TRUE' }
VERSION : 0.1
// test
// stored: AutoNumber true, UDAEnableTagReadback false
BEGIN

NETWORK
TITLE = Main
// comment: PLC1
      CALL  "BST_VALVE_400", "DB";


//Call the CM FB with the corresponding DB instance
END_FUNCTION

FUNCTION "MV006_fc" : Void   // FC1, STL
TITLE = MV006_fc
{ S7_Optimized_Access := 'TRUE' }
VERSION : 0.1
// test
// stored: AutoNumber true, UDAEnableTagReadback false
BEGIN

NETWORK
TITLE = Main
// comment: PLC1
      CALL  "BST_VALVE_400", "DB";


//Call the CM FB with the corresponding DB instance
END_FUNCTION

FUNCTION "MV007_fc" : Void   // FC1, STL
TITLE = MV007_fc
{ S7_Optimized_Access := 'TRUE' }
VERSION : 0.1
// test
// stored: AutoNumber true, UDAEnableTagReadback false
BEGIN

NETWORK
TITLE = Main
// comment: PLC1
      CALL  "BST_VALVE_400", "DB";


//Call the CM FB with the corresponding DB instance
END_FUNCTION

FUNCTION "P100_fc" : Void   // FC1, STL
TITLE = P100_fc
{ S7_Optimized_Access := 'TRUE' }
VERSION : 0.1
// test
// stored: AutoNumber true, UDAEnableTagReadback false
BEGIN

NETWORK
TITLE = Main
// comment: PLC1
      CALL  "BST_VALVE_400", "DB";


//Call the CM FB with the corresponding DB instance
END_FUNCTION

FUNCTION "P101_fc" : Void   // FC1, STL
TITLE = P101_fc
{ S7_Optimized_Access := 'TRUE' }
VERSION : 0.1
// test
// stored: AutoNumber true, UDAEnableTagReadback false
BEGIN

NETWORK
TITLE = Main
// comment: PLC1
      CALL  "BST_MOTOR_400", "DB";


//Call the CM FB with the corresponding DB instance
END_FUNCTION

FUNCTION "P200_fc" : Void   // FC1, STL
TITLE = P200_fc
{ S7_Optimized_Access := 'TRUE' }
VERSION : 0.1
// test
// stored: AutoNumber true, UDAEnableTagReadback false
BEGIN

NETWORK
TITLE = Main
// comment: PLC1
      CALL  "BST_MOTOR_400", "DB";


//Call the CM FB with the corresponding DB instance
END_FUNCTION

FUNCTION "P201_fc" : Void   // FC1, STL
TITLE = P201_fc
{ S7_Optimized_Access := 'TRUE' }
VERSION : 0.1
// test
// stored: AutoNumber true, UDAEnableTagReadback false
BEGIN

NETWORK
TITLE = Main
// comment: PLC1
      CALL  "BST_MOTOR_400", "DB";


//Call the CM FB with the corresponding DB instance
END_FUNCTION

FUNCTION "T100_fc" : Void   // FC1, STL
TITLE = _fc
{ S7_Optimized_Access := 'TRUE' }
VERSION : 0.1
// test
// stored: AutoNumber true, UDAEnableTagReadback false
BEGIN

NETWORK
TITLE = Main


// code


END_FUNCTION

FUNCTION "T101_fc" : Void   // FC1, STL
TITLE = _fc
{ S7_Optimized_Access := 'TRUE' }
VERSION : 0.1
// test
// stored: AutoNumber true, UDAEnableTagReadback false
BEGIN

NETWORK
TITLE = Main


// code


END_FUNCTION

FUNCTION "T102_fc" : Void   // FC1, STL
TITLE = _fc
{ S7_Optimized_Access := 'TRUE' }
VERSION : 0.1
// test
// stored: AutoNumber true, UDAEnableTagReadback false
BEGIN

NETWORK
TITLE = Main


// code


END_FUNCTION

FUNCTION "T103_fc" : Void   // FC1, STL
TITLE = _fc
{ S7_Optimized_Access := 'TRUE' }
VERSION : 0.1
// test
// stored: AutoNumber true, UDAEnableTagReadback false
BEGIN

NETWORK
TITLE = Main


// code


END_FUNCTION

FUNCTION "T104_fc" : Void   // FC1, STL
TITLE = _fc
{ S7_Optimized_Access := 'TRUE' }
VERSION : 0.1
// test
// stored: AutoNumber true, UDAEnableTagReadback false
BEGIN

NETWORK
TITLE = Main


// code


END_FUNCTION

FUNCTION "T105_fc" : Void   // FC1, STL
TITLE = _fc
{ S7_Optimized_Access := 'TRUE' }
VERSION : 0.1
// test
// stored: AutoNumber true, UDAEnableTagReadback false
BEGIN

NETWORK
TITLE = Main


// code


END_FUNCTION

FUNCTION "T106_fc" : Void   // FC1, STL
TITLE = _fc
{ S7_Optimized_Access := 'TRUE' }
VERSION : 0.1
// test
// stored: AutoNumber true, UDAEnableTagReadback false
BEGIN

NETWORK
TITLE = Main


// code


END_FUNCTION

FUNCTION "T107_fc" : Void   // FC1, STL
TITLE = _fc
{ S7_Optimized_Access := 'TRUE' }
VERSION : 0.1
// test
// stored: AutoNumber true, UDAEnableTagReadback false
BEGIN

NETWORK
TITLE = Main


// code


END_FUNCTION

FUNCTION "T108_fc" : Void   // FC1, STL
TITLE = _fc
{ S7_Optimized_Access := 'TRUE' }
VERSION : 0.1
// test
// stored: AutoNumber true, UDAEnableTagReadback false
BEGIN

NETWORK
TITLE = Main


// code


END_FUNCTION

FUNCTION "T109_fc" : Void   // FC1, STL
TITLE = _fc
{ S7_Optimized_Access := 'TRUE' }
VERSION : 0.1
// test
// stored: AutoNumber true, UDAEnableTagReadback false
BEGIN

NETWORK
TITLE = Main


// code


END_FUNCTION

FUNCTION "T110_fc" : Void   // FC1, STL
TITLE = _fc
{ S7_Optimized_Access := 'TRUE' }
VERSION : 0.1
// test
// stored: AutoNumber true, UDAEnableTagReadback false
BEGIN

NETWORK
TITLE = Main


// code


END_FUNCTION

FUNCTION "T111_fc" : Void   // FC1, STL
TITLE = _fc
{ S7_Optimized_Access := 'TRUE' }
VERSION : 0.1
// test
// stored: AutoNumber true, UDAEnableTagReadback false
BEGIN

NETWORK
TITLE = Main


// code


END_FUNCTION

FUNCTION "T112_fc" : Void   // FC1, STL
TITLE = _fc
{ S7_Optimized_Access := 'TRUE' }
VERSION : 0.1
// test
// stored: AutoNumber true, UDAEnableTagReadback false
BEGIN

NETWORK
TITLE = Main


// code


END_FUNCTION

FUNCTION "T113_fc" : Void   // FC1, STL
TITLE = _fc
{ S7_Optimized_Access := 'TRUE' }
VERSION : 0.1
// test
// stored: AutoNumber true, UDAEnableTagReadback false
BEGIN

NETWORK
TITLE = Main


// code


END_FUNCTION

FUNCTION "T114_fc" : Void   // FC1, STL
TITLE = _fc
{ S7_Optimized_Access := 'TRUE' }
VERSION : 0.1
// test
// stored: AutoNumber true, UDAEnableTagReadback false
BEGIN

NETWORK
TITLE = Main


// code


END_FUNCTION

FUNCTION "XV001_fc" : Void   // FC1, STL
TITLE = XV001_fc
{ S7_Optimized_Access := 'TRUE' }
VERSION : 0.1
// Some Valve  on drawing 1 test
// stored: AutoNumber true, UDAEnableTagReadback false
BEGIN

NETWORK
TITLE = Main
// comment: PLC1


//Call the CM FB with the corresponding DB instance
END_FUNCTION

FUNCTION "XV002_fc" : Void   // FC1, STL
TITLE = XV002_fc
{ S7_Optimized_Access := 'TRUE' }
VERSION : 0.1
// Some Valve  on drawing 2 test
// stored: AutoNumber true, UDAEnableTagReadback false
BEGIN

NETWORK
TITLE = Main
// comment: PLC1


// Call the CM FB with the corresponding DB instance
      CALL  "BST_VALVE_400", "XV002"
      ( AUT_OP   := ,
        FB_OPEN  := ,
        FB_CLOSE := ,
        QOPEN    := ,
        QCLOSE   := ,
        QMON_ERR := ,
        QCMD_OP  := 
      );
END_FUNCTION

FUNCTION "XV003_fc" : Void   // FC1, STL
TITLE = XV003_fc
{ S7_Optimized_Access := 'TRUE' }
VERSION : 0.1
// Some Valve  on drawing 3 test
// stored: AutoNumber true, UDAEnableTagReadback false
BEGIN

NETWORK
TITLE = Main
// comment: PLC1
      CALL  "BST_VALVE_400", "DB";


//Call the CM FB with the corresponding DB instance
END_FUNCTION

FUNCTION "XV004_fc" : Void   // FC1, STL
TITLE = XV004_fc
{ S7_Optimized_Access := 'TRUE' }
VERSION : 0.1
// Some Valve  on drawing 4 test
// stored: AutoNumber true, UDAEnableTagReadback false
BEGIN

NETWORK
TITLE = Main
// comment: PLC1
      CALL  "BST_VALVE_400", "DB";


//Call the CM FB with the corresponding DB instance
END_FUNCTION

FUNCTION "XV300_fc" : Void   // FC1, STL
TITLE = XV300_fc
{ S7_Optimized_Access := 'TRUE' }
VERSION : 0.1
// Some Valve  on drawing 15 test
// stored: AutoNumber true, UDAEnableTagReadback false
BEGIN

NETWORK
TITLE = Main
// comment: PLC1
      CALL  "BST_VALVE_400", "DB";


//Call the CM FB with the corresponding DB instance
END_FUNCTION

FUNCTION "XV301_fc" : Void   // FC1, STL
TITLE = XV301_fc
{ S7_Optimized_Access := 'TRUE' }
VERSION : 0.1
// Some Valve  on drawing 18 test
// stored: AutoNumber true, UDAEnableTagReadback false
BEGIN

NETWORK
TITLE = Main
// comment: PLC1
      CALL  "BST_VALVE_400", "DB";


//Call the CM FB with the corresponding DB instance
END_FUNCTION

FUNCTION "XV400_fc" : Void   // FC1, STL
TITLE = XV400_fc
{ S7_Optimized_Access := 'TRUE' }
VERSION : 0.1
// Some Valve  on drawing 16 test
// stored: AutoNumber true, UDAEnableTagReadback false
BEGIN

NETWORK
TITLE = Main
// comment: PLC1
      CALL  "BST_VALVE_400", "DB";


//Call the CM FB with the corresponding DB instance
END_FUNCTION

FUNCTION "XV401_fc" : Void   // FC1, STL
TITLE = XV401_fc
{ S7_Optimized_Access := 'TRUE' }
VERSION : 0.1
// Some Valve  on drawing 21 test
// stored: AutoNumber true, UDAEnableTagReadback false
BEGIN

NETWORK
TITLE = Main
// comment: PLC1
      CALL  "BST_VALVE_400", "DB";


//Call the CM FB with the corresponding DB instance
END_FUNCTION

FUNCTION "XV500_fc" : Void   // FC1, STL
TITLE = XV500_fc
{ S7_Optimized_Access := 'TRUE' }
VERSION : 0.1
// Some Valve  on drawing 17 test
// stored: AutoNumber true, UDAEnableTagReadback false
BEGIN

NETWORK
TITLE = Main
// comment: PLC1
      CALL  "BST_VALVE_400", "DB";


//Call the CM FB with the corresponding DB instance
END_FUNCTION

FUNCTION "XV501_fc" : Void   // FC1, STL
TITLE = XV501_fc
{ S7_Optimized_Access := 'TRUE' }
VERSION : 0.1
// Some Valve  on drawing 20 test
// stored: AutoNumber true, UDAEnableTagReadback false
BEGIN

NETWORK
TITLE = Main
// comment: PLC1
      CALL  "BST_VALVE_400", "DB";


//Call the CM FB with the corresponding DB instance
END_FUNCTION

FUNCTION "em_read" : Void   // FC1, STL
{ S7_Optimized_Access := 'TRUE' }
VERSION : 0.1
// stored: AutoNumber true, UDAEnableTagReadback false
   VAR_INPUT
      EM_ID : Int;
      UDT_LOCATION : Pointer;
      UDT_OFFSET : Int;
      Length : Int;
   END_VAR
   VAR_OUTPUT
      EM_addressing_error : Bool;
   END_VAR
   VAR_TEMP
      em_address : Int;
      em_index_length : Int;
      em_db : Int;
      em_udt : Int;
      phase_db : Int;
      phase_udt : Int;
      source_pointer : Any;
      dest_pointer : Any;
      blkmov_retval : Int;
   END_VAR
BEGIN

NETWORK
TITLE = 

// Calculate the amount of EMs in the EM_Index

      OPN   "EM_Index";
      L     DBLG;
      L     4;
      /I;
      T     #em_index_length;

// protect against an address outside db25
      L     #EM_ID;
      L     #em_index_length;
      >I;
      =     #EM_addressing_error;
      JC    ENDS;


// calculate the address of the EM in DB25
      L     #EM_ID;
      L     4;
      *I;
      T     #em_address;

// prepare the pointer for the location in EM Index DB
// todo: probably don't need to load the 0-pointer
      L     P#DBX0.0;
      L     #em_address;
      SLD   3;
      +D;
      LAR1;

// read the DB number
      L     DBW [AR1, P#0.0];
      T     #em_db;

// read the UDT location
      L     DBW [AR1, P#2.0];
      T     #em_udt;

// read the start of the UDT in the phase
      L     P##UDT_LOCATION;
      LAR1;
      L     D [AR1, P#2.0];
      L     DW#16#7FFF8;
      AD;
      SRD   3;
      T     #phase_udt;

// read the phase DB
      L     W [AR1, P#0.0];
      T     #phase_db;

// prepare the sending address
      LAR1  P##source_pointer;
      L     W#16#1002;  //Syntax ID (10h for S7, 2h bytes)
      T     W [AR1, P#0.0];
      L     #Length;  //Length in bytes
      T     W [AR1, P#2.0];
      L     #em_db;  //DB-nummer EM
      T     W [AR1, P#4.0];
      L     #em_udt;  //Start address in DB EM
      L     #UDT_OFFSET;
      +I;
      SLD   3;
      L     DW#16#84000000;
      OD;
      T     D [AR1, P#6.0];

// prepare the receiving address
      LAR1  P##dest_pointer;
      L     W#16#1002;  //Syntax ID (10h for S7, 2h bytes)
      T     W [AR1, P#0.0];
      L     #Length;  //Length in bytes
      T     W [AR1, P#2.0];
      L     #phase_db;  //DB-nummer SEQ
      T     W [AR1, P#4.0];
      L     #phase_udt;  //Start address in DB SEQ
      L     #UDT_OFFSET;
      +I;
      SLD   3;
      L     DW#16#84000000;
      OD;
      T     D [AR1, P#6.0];

// copy the data
      CALL  BLKMOV
      ( SRCBLK  := #source_pointer,
        RET_VAL := #blkmov_retval,
        DSTBLK  := #dest_pointer
      );




ENDS: NOP   0;


END_FUNCTION

FUNCTION "em_write" : Void   // FC1, STL
{ S7_Optimized_Access := 'FALSE' }
VERSION : 0.1
// stored: AutoNumber true, UDAEnableTagReadback false
   VAR_INPUT
      EM_ID : Int;
      UDT_LOCATION : Pointer;
      UDT_OFFSET : Int;
      Length : Int;
      Request : Int;
      Owner : Int;
   END_VAR
   VAR_OUTPUT
      EM_addressing_error : Bool;
   END_VAR
   VAR_TEMP
      em_address : Int;
      em_index_length : Int;
      em_db : Int;
      em_udt : Int;
      phase_db : Int;
      phase_udt : Int;
      source_pointer : Any;
      dest_pointer : Any;
      adjusted_length : Int;
      blkmov_retval : Int;
   END_VAR
BEGIN

NETWORK
TITLE = 

// Skip the entire FC if Request = 0

      L     #Request;
      L     0;
      ==I;
      JCN   ENDS;

// Reduce the length to one Integer if the EM has not been acquired yet
      L     #Owner;
      L     #Request;
      <>I;
      JCN   REDU;

      L     2;
      T     #adjusted_length;

REDU: NOP   0;


// Calculate the amount of EMs in the EM_Index
      OPN   "db25";
      L     DBLG;
      L     4;
      /I;
      T     #em_index_length;


// protect against an address outside db25
      L     #EM_ID;
      L     #em_index_length;
      >I;
      =     #EM_addressing_error;
      JC    ENDS;


// calculate the address of the EM in DB25
      L     #EM_ID;
      L     4;
      *I;
      T     #em_address;

// prepare the pointer for the location in EM Index DB
// todo: probably don't need to load the 0-pointer
      L     P#DBX0.0;
      L     #em_address;
      SLD   3;
      +D;
      LAR1;

// read the DB number
      L     DBW [AR1, P#0.0];
      T     #em_db;

// read the UDT location
      L     DBW [AR1, P#2.0];
      T     #em_udt;

// read the start of the UDT in the phase
      L     P##UDT_LOCATION;
      LAR1;
      L     DBD [AR1, P#2.0];
      L     DW#16#7FFF8;
      AD;
      SRD   3;
      T     #phase_udt;

// read the phase DB
      L     DBW [AR1, P#0.0];
      T     #phase_db;

// prepare the receiving address
      LAR1  P##dest_pointer;
      L     W#16#1002;  //Syntax ID (10h for S7, 2h bytes)
      T     DBW [AR1, P#0.0];
      L     #adjusted_length;  //Length in bytes
      T     DBW [AR1, P#2.0];
      L     #em_db;  //DB-nummer EM
      T     DBW [AR1, P#4.0];
      L     #em_udt;  //Start address in DB EM
      L     #UDT_OFFSET;
      +I;
      SLD   3;
      L     DW#16#84000000;
      OD;
      T     DBD [AR1, P#6.0];

// prepare the sending address
      LAR1  P##source_pointer;
      L     W#16#1002;  //Syntax ID (10h for S7, 2h bytes)
      T     DBW [AR1, P#0.0];
      L     #adjusted_length;  //Length in bytes
      T     DBW [AR1, P#2.0];
      L     #phase_db;  //DB-nummer SEQ
      T     DBW [AR1, P#4.0];
      L     #phase_udt;  //Start address in DB SEQ
      L     #UDT_OFFSET;
      +I;
      SLD   3;
      L     DW#16#84000000;
      OD;
      T     DBD [AR1, P#6.0];

// copy the data
      CALL  BLKMOV
      ( SRCBLK  := #source_pointer,
        RET_VAL := #blkmov_retval,
        DSTBLK  := #dest_pointer
      );




ENDS: NOP   0;


END_FUNCTION

FUNCTION "Control_Modules" : Void   // FC1, STL
TITLE = Program
{ S7_Optimized_Access := 'TRUE' }
VERSION : 0.1
// Call all the Control Modules
// stored: AutoNumber true, UDAEnableTagReadback false
BEGIN

NETWORK
TITLE = Main
// comment

      CALL  "FIC101_fc";



END_FUNCTION

FUNCTION "Equipment_Modules" : Void   // FC1, STL
TITLE = Program
{ S7_Optimized_Access := 'TRUE' }
VERSION : 0.1
// Call all the Equipment Modules
// stored: AutoNumber true, UDAEnableTagReadback false
BEGIN

NETWORK
TITLE = Main
// comment

      CALL  "EM_Instance_14_fc";



END_FUNCTION

FUNCTION "Phases" : Void   // FC1, STL
TITLE = Program
{ S7_Optimized_Access := 'TRUE' }
VERSION : 0.1
// Call all the Phases
// stored: AutoNumber true, UDAEnableTagReadback false
BEGIN

NETWORK
TITLE = Main
// comment

      CALL  "phase_2_fc";



END_FUNCTION

FUNCTION "phase_2_fc" : Void   // FC1, STL
TITLE = _fc
{ S7_Optimized_Access := 'TRUE' }
VERSION : 0.1
// Second instance of fds_example test
// stored: AutoNumber true, UDAEnableTagReadback false
BEGIN

NETWORK
TITLE = Main
// comment: Second instance of fds_example


